C03661=1165.094,157.348,-57.134,-178.430,6.708,148.774
C03662=1165.089,157.596,-57.156,-178.428,6.710,148.774
C03663=1165.084,157.866,-57.179,-178.425,6.712,148.774
C03664=1165.079,158.135,-57.202,-178.422,6.714,148.773
C03665=1165.073,158.404,-57.226,-178.419,6.716,148.773
C03666=1165.069,158.672,-57.249,-178.416,6.718,148.772
C03667=1165.064,158.922,-57.270,-178.414,6.720,148.772
C03668=1165.059,159.170,-57.292,-178.411,6.721,148.772
C03669=1165.055,159.420,-57.314,-178.408,6.723,148.771
C03670=1165.050,159.668,-57.335,-178.405,6.725,148.771
C03671=1165.045,159.918,-57.356,-178.403,6.727,148.771
C03672=1165.040,160.167,-57.378,-178.399,6.729,148.770
C03673=1165.035,160.416,-57.400,-178.397,6.731,148.770
C03674=1165.031,160.664,-57.422,-178.395,6.733,148.770
C03675=1165.026,160.914,-57.444,-178.392,6.735,148.769
C03676=1165.021,161.163,-57.465,-178.389,6.737,148.769
C03677=1165.017,161.412,-57.487,-178.386,6.738,148.769
C03678=1165.012,161.661,-57.509,-178.384,6.740,148.768
C03679=1165.007,161.909,-57.530,-178.381,6.742,148.768
C03680=1165.003,162.159,-57.552,-178.378,6.744,148.767
C03681=1164.998,162.407,-57.574,-178.375,6.746,148.767
C03682=1164.994,162.657,-57.596,-178.372,6.748,148.767
C03683=1164.989,162.906,-57.617,-178.370,6.750,148.766
C03684=1164.984,163.155,-57.639,-178.367,6.751,148.766
C03685=1164.979,163.404,-57.661,-178.364,6.753,148.766
C03686=1164.975,163.653,-57.682,-178.362,6.755,148.765
C03687=1164.970,163.902,-57.704,-178.359,6.757,148.765
C03688=1164.965,164.151,-57.726,-178.357,6.759,148.765
C03689=1164.961,164.400,-57.748,-178.353,6.761,148.764
C03690=1164.956,164.649,-57.770,-178.351,6.763,148.764
C03691=1164.951,164.897,-57.792,-178.348,6.765,148.764
C03692=1164.947,165.147,-57.814,-178.345,6.767,148.763
C03693=1164.942,165.395,-57.835,-178.343,6.768,148.763
C03694=1164.937,165.645,-57.858,-178.340,6.770,148.762
C03695=1164.932,165.893,-57.880,-178.337,6.772,148.762
C03696=1164.928,166.143,-57.902,-178.335,6.775,148.762
C03697=1164.923,166.391,-57.923,-178.332,6.776,148.762
C03698=1164.919,166.641,-57.945,-178.329,6.778,148.761
C03699=1164.914,166.889,-57.967,-178.326,6.780,148.761
C03700=1164.910,167.139,-57.989,-178.324,6.782,148.760
C03701=1164.905,167.387,-58.012,-178.321,6.783,148.760
C03702=1164.900,167.636,-58.034,-178.318,6.786,148.760
C03703=1164.895,167.885,-58.056,-178.315,6.788,148.759
C03704=1164.891,168.134,-58.078,-178.313,6.790,148.759
C03705=1164.886,168.383,-58.100,-178.310,6.792,148.759
C03706=1164.881,168.633,-58.122,-178.308,6.793,148.758
C03707=1164.876,168.881,-58.144,-178.305,6.795,148.758
C03708=1164.872,169.130,-58.167,-178.302,6.798,148.758
C03709=1164.868,169.379,-58.188,-178.299,6.799,148.757
C03710=1164.863,169.628,-58.211,-178.296,6.801,148.757
C03711=1164.858,169.877,-58.233,-178.294,6.803,148.757
C03712=1164.853,170.126,-58.255,-178.291,6.805,148.757
C03713=1164.849,170.375,-58.277,-178.289,6.807,148.756
C03714=1164.844,170.624,-58.300,-178.285,6.809,148.756
C03715=1164.840,170.873,-58.322,-178.283,6.811,148.755
C03716=1164.835,171.122,-58.343,-178.280,6.813,148.755
C03717=1164.830,171.371,-58.367,-178.277,6.815,148.755
C03718=1164.825,171.620,-58.388,-178.275,6.817,148.755
C03719=1164.821,171.869,-58.411,-178.272,6.819,148.754
C03720=1164.816,172.118,-58.434,-178.269,6.821,148.754
C03721=1164.811,172.367,-58.456,-178.266,6.823,148.753
C03722=1164.807,172.616,-58.478,-178.264,6.825,148.753
C03723=1164.802,172.864,-58.501,-178.261,6.826,148.753
C03724=1164.797,173.114,-58.523,-178.258,6.829,148.753
C03725=1164.793,173.363,-58.545,-178.256,6.831,148.752
C03726=1164.788,173.611,-58.568,-178.253,6.833,148.752
C03727=1164.784,173.861,-58.590,-178.250,6.835,148.752
C03728=1164.780,174.109,-58.613,-178.248,6.836,148.751
C03729=1164.774,174.358,-58.635,-178.244,6.839,148.751
C03730=1164.770,174.608,-58.657,-178.242,6.841,148.751
C03731=1164.764,174.856,-58.680,-178.239,6.843,148.750
C03732=1164.760,175.105,-58.702,-178.237,6.845,148.750
C03733=1164.756,175.354,-58.725,-178.234,6.846,148.750
C03734=1164.751,175.603,-58.747,-178.231,6.849,148.749
C03735=1164.747,175.852,-58.770,-178.228,6.851,148.749
C03736=1164.742,176.101,-58.792,-178.226,6.853,148.749
C03737=1164.737,176.349,-58.815,-178.223,6.854,148.748
C03738=1164.732,176.599,-58.837,-178.220,6.857,148.748
C03739=1164.728,176.848,-58.860,-178.217,6.859,148.748
C03740=1164.723,177.098,-58.883,-178.214,6.861,148.747
C03741=1164.719,177.346,-58.905,-178.212,6.863,148.747
C03742=1164.714,177.595,-58.928,-178.210,6.864,148.747
C03743=1164.710,177.844,-58.951,-178.206,6.867,148.746
C03744=1164.704,178.092,-58.974,-178.204,6.869,148.746
C03745=1164.700,178.342,-58.996,-178.201,6.870,148.746
C03746=1164.695,178.591,-59.019,-178.199,6.873,148.746
C03747=1164.691,178.839,-59.042,-178.195,6.875,148.745
C03748=1164.686,179.088,-59.064,-178.193,6.877,148.745
C03749=1164.682,179.337,-59.087,-178.190,6.879,148.745
C03750=1164.677,179.587,-59.109,-178.188,6.881,148.744
C03751=1164.672,179.835,-59.132,-178.185,6.883,148.744
C03752=1164.668,180.084,-59.155,-178.182,6.885,148.744
C03753=1164.663,180.333,-59.179,-178.179,6.887,148.743
C03754=1164.659,180.582,-59.201,-178.177,6.889,148.743
C03755=1164.654,180.831,-59.224,-178.174,6.892,148.743
C03756=1164.649,181.079,-59.246,-178.171,6.893,148.742
C03757=1164.645,181.328,-59.270,-178.168,6.895,148.742
C03758=1164.640,181.578,-59.292,-178.166,6.897,148.742
C03759=1164.636,181.827,-59.315,-178.163,6.900,148.742
C03760=1164.630,182.075,-59.338,-178.160,6.902,148.741
C03761=1164.626,182.324,-59.361,-178.158,6.903,148.741
C03762=1164.621,182.573,-59.384,-178.154,6.906,148.741
C03763=1164.617,182.822,-59.407,-178.152,6.908,148.740
C03764=1164.613,183.071,-59.430,-178.149,6.910,148.740
C03765=1164.607,183.319,-59.453,-178.147,6.912,148.740
C03766=1164.603,183.568,-59.476,-178.144,6.914,148.739
C03767=1164.598,183.838,-59.500,-178.141,6.916,148.739
C03768=1164.593,184.108,-59.525,-178.138,6.919,148.739
C03769=1164.588,184.377,-59.551,-178.135,6.921,148.739
C03770=1164.583,184.647,-59.575,-178.132,6.923,148.738
C03771=1164.578,184.896,-59.598,-178.129,6.925,148.738
C03772=1164.574,185.145,-59.622,-178.127,6.927,148.738
C03773=1164.569,185.394,-59.645,-178.124,6.930,148.737
C03774=1164.565,185.643,-59.668,-178.121,6.931,148.737
C03775=1164.560,185.892,-59.691,-178.119,6.933,148.737
C03776=1164.555,186.141,-59.715,-178.115,6.936,148.736
C03777=1164.551,186.390,-59.738,-178.113,6.938,148.736
C03778=1164.546,186.638,-59.760,-178.110,6.940,148.736
C03779=1164.541,186.887,-59.784,-178.108,6.941,148.735
C03780=1164.537,187.136,-59.807,-178.104,6.944,148.735
C03781=1164.532,187.385,-59.830,-178.102,6.946,148.735
C03782=1164.527,187.634,-59.854,-178.100,6.948,148.735
C03783=1164.523,187.883,-59.876,-178.096,6.950,148.734
C03784=1164.519,188.132,-59.900,-178.094,6.952,148.734
C03785=1164.514,188.381,-59.923,-178.091,6.954,148.734
C03786=1164.509,188.630,-59.947,-178.088,6.957,148.734
C03787=1164.505,188.878,-59.971,-178.086,6.959,148.733
C03788=1164.500,189.126,-59.994,-178.083,6.961,148.733
C03789=1164.495,189.375,-60.017,-178.080,6.963,148.733
C03790=1164.491,189.624,-60.040,-178.077,6.965,148.732
C03791=1164.486,189.873,-60.063,-178.075,6.967,148.732
C03792=1164.482,190.122,-60.086,-178.072,6.970,148.732
C03793=1164.477,190.371,-60.110,-178.069,6.971,148.732
C03794=1164.472,190.620,-60.134,-178.067,6.974,148.731
C03795=1164.468,190.869,-60.157,-178.064,6.976,148.731
C03796=1164.463,191.118,-60.181,-178.061,6.978,148.731
C03797=1164.458,191.367,-60.204,-178.058,6.980,148.730
C03798=1164.454,191.616,-60.227,-178.056,6.983,148.730
C03799=1164.449,191.864,-60.251,-178.053,6.984,148.730
C03800=1164.445,192.113,-60.275,-178.050,6.986,148.730
C03801=1164.440,192.362,-60.298,-178.047,6.989,148.729
C03802=1164.435,192.611,-60.322,-178.045,6.991,148.729
C03803=1164.431,192.860,-60.346,-178.042,6.993,148.729
C03804=1164.426,193.109,-60.369,-178.039,6.996,148.729
C03805=1164.421,193.358,-60.392,-178.037,6.997,148.728
C03806=1164.417,193.606,-60.416,-178.034,6.999,148.728
C03807=1164.412,193.855,-60.440,-178.031,7.002,148.728
C03808=1164.408,194.104,-60.464,-178.029,7.004,148.727
C03809=1164.403,194.353,-60.487,-178.026,7.006,148.727
C03810=1164.399,194.602,-60.510,-178.023,7.008,148.727
C03811=1164.394,194.850,-60.535,-178.020,7.010,148.727
C03812=1164.389,195.099,-60.558,-178.018,7.012,148.726
C03813=1164.385,195.348,-60.581,-178.015,7.015,148.726
C03814=1164.380,195.597,-60.605,-178.012,7.017,148.726
C03815=1164.376,195.846,-60.629,-178.009,7.019,148.725
C03816=1164.371,196.094,-60.653,-178.007,7.021,148.725
C03817=1164.367,196.344,-60.677,-178.004,7.023,148.725
C03818=1164.363,196.592,-60.701,-178.001,7.026,148.725
C03819=1164.358,196.841,-60.724,-177.999,7.028,148.725
C03820=1164.353,197.090,-60.749,-177.996,7.030,148.724
C03821=1164.348,197.339,-60.772,-177.993,7.033,148.724
C03822=1164.344,197.587,-60.796,-177.991,7.034,148.724
C03823=1164.339,197.836,-60.819,-177.987,7.037,148.723
C03824=1164.335,198.085,-60.843,-177.985,7.039,148.723
C03825=1164.330,198.334,-60.867,-177.982,7.041,148.723
C03826=1164.326,198.582,-60.891,-177.979,7.043,148.723
C03827=1164.321,198.832,-60.916,-177.977,7.046,148.722
C03828=1164.316,199.081,-60.939,-177.974,7.047,148.722
C03829=1164.312,199.329,-60.963,-177.971,7.050,148.722
C03830=1164.307,199.578,-60.987,-177.969,7.052,148.722
C03831=1164.303,199.827,-61.011,-177.966,7.055,148.721
C03832=1164.299,200.075,-61.035,-177.963,7.057,148.721
C03833=1164.294,200.325,-61.059,-177.961,7.058,148.721
C03834=1164.289,200.574,-61.083,-177.958,7.061,148.721
C03835=1164.285,200.822,-61.107,-177.955,7.063,148.720
C03836=1164.280,201.071,-61.131,-177.952,7.066,148.720
C03837=1164.275,201.320,-61.155,-177.950,7.068,148.720
C03838=1164.271,201.568,-61.179,-177.947,7.070,148.720
C03839=1164.267,201.817,-61.204,-177.944,7.072,148.719
C03840=1164.262,202.066,-61.227,-177.942,7.074,148.719
C03841=1164.257,202.315,-61.252,-177.938,7.077,148.719
C03842=1164.253,202.563,-61.276,-177.936,7.079,148.719
C03843=1164.248,202.812,-61.300,-177.933,7.082,148.718
C03844=1164.243,203.062,-61.324,-177.931,7.084,148.718
C03845=1164.239,203.310,-61.348,-177.928,7.086,148.718
C03846=1164.235,203.559,-61.373,-177.925,7.088,148.718
C03847=1164.229,203.807,-61.397,-177.923,7.090,148.717
C03848=1164.226,204.056,-61.422,-177.919,7.093,148.717
C03849=1164.221,204.305,-61.446,-177.917,7.095,148.717
C03850=1164.216,204.554,-61.470,-177.914,7.097,148.717
C03851=1164.211,204.803,-61.494,-177.911,7.099,148.716
C03852=1164.208,205.052,-61.518,-177.909,7.101,148.716
C03853=1164.203,205.300,-61.543,-177.906,7.104,148.716
C03854=1164.198,205.549,-61.567,-177.904,7.106,148.716
C03855=1164.194,205.797,-61.591,-177.900,7.109,148.715
C03856=1164.189,206.047,-61.616,-177.898,7.111,148.715
C03857=1164.185,206.295,-61.640,-177.895,7.113,148.715
C03858=1164.180,206.544,-61.665,-177.893,7.116,148.715
C03859=1164.175,206.792,-61.689,-177.890,7.117,148.715
C03860=1164.171,207.042,-61.714,-177.887,7.120,148.714
C03861=1164.166,207.290,-61.738,-177.885,7.122,148.714
C03862=1164.161,207.539,-61.763,-177.881,7.125,148.714
C03863=1164.157,207.788,-61.787,-177.879,7.127,148.714
C03864=1164.153,208.036,-61.811,-177.876,7.129,148.713
C03865=1164.148,208.285,-61.836,-177.874,7.131,148.713
C03866=1164.144,208.533,-61.860,-177.870,7.134,148.713
C03867=1164.139,208.783,-61.885,-177.868,7.136,148.713
C03868=1164.135,209.031,-61.909,-177.865,7.139,148.712
C03869=1164.129,209.280,-61.934,-177.863,7.141,148.712
C03870=1164.126,209.529,-61.958,-177.860,7.143,148.712
C03871=1164.121,209.799,-61.985,-177.857,7.145,148.712
C03872=1164.116,210.070,-62.012,-177.854,7.148,148.712
C03873=1164.111,210.340,-62.039,-177.851,7.151,148.711
C03874=1164.106,210.611,-62.065,-177.848,7.153,148.711
C03875=1164.101,210.860,-62.090,-177.845,7.155,148.711
C03876=1164.096,211.109,-62.115,-177.842,7.158,148.711
C03877=1164.092,211.358,-62.140,-177.840,7.160,148.710
C03878=1164.087,211.606,-62.165,-177.837,7.162,148.710
C03879=1164.083,211.854,-62.189,-177.834,7.165,148.710
C03880=1164.078,212.104,-62.214,-177.832,7.167,148.710
C03881=1164.073,212.352,-62.239,-177.829,7.170,148.710
C03882=1164.069,212.600,-62.263,-177.826,7.171,148.709
C03883=1164.065,212.850,-62.288,-177.824,7.174,148.709
C03884=1164.060,213.098,-62.313,-177.821,7.176,148.709
C03885=1164.056,213.348,-62.338,-177.818,7.179,148.709
C03886=1164.051,213.596,-62.363,-177.815,7.181,148.708
C03887=1164.047,213.845,-62.387,-177.813,7.184,148.708
C03888=1164.042,214.093,-62.412,-177.810,7.186,148.708
C03889=1164.037,214.342,-62.437,-177.807,7.189,148.708
C03890=1164.033,214.591,-62.462,-177.805,7.190,148.707
C03891=1164.028,214.839,-62.487,-177.802,7.193,148.707
C03892=1164.024,215.088,-62.512,-177.799,7.195,148.707
C03893=1164.020,215.337,-62.536,-177.796,7.198,148.707
C03894=1164.015,215.585,-62.562,-177.794,7.200,148.707
C03895=1164.010,215.834,-62.587,-177.791,7.203,148.707
C03896=1164.006,216.084,-62.612,-177.788,7.204,148.706
C03897=1164.002,216.331,-62.637,-177.785,7.207,148.706
C03898=1163.997,216.581,-62.662,-177.783,7.209,148.706
C03899=1163.992,216.829,-62.687,-177.780,7.212,148.706
C03900=1163.988,217.078,-62.712,-177.777,7.215,148.706
C03901=1163.984,217.326,-62.737,-177.775,7.217,148.705
C03902=1163.979,217.576,-62.762,-177.772,7.220,148.705
C03903=1163.974,217.824,-62.787,-177.769,7.222,148.705
C03904=1163.970,218.073,-62.812,-177.766,7.224,148.705
C03905=1163.965,218.321,-62.838,-177.764,7.226,148.704
C03906=1163.961,218.570,-62.862,-177.761,7.229,148.704
C03907=1163.956,218.818,-62.888,-177.758,7.231,148.704
C03908=1163.952,219.067,-62.913,-177.756,7.234,148.704
C03909=1163.947,219.316,-62.938,-177.753,7.236,148.704
C03910=1163.943,219.565,-62.964,-177.750,7.239,148.703
C03911=1163.938,219.814,-62.989,-177.748,7.241,148.703
C03912=1163.934,220.062,-63.014,-177.745,7.243,148.703
C03913=1163.930,220.311,-63.039,-177.742,7.246,148.703
C03914=1163.925,220.559,-63.064,-177.739,7.248,148.703
C03915=1163.921,220.808,-63.090,-177.736,7.251,148.703
C03916=1163.916,221.056,-63.115,-177.734,7.253,148.702
C03917=1163.911,221.306,-63.140,-177.731,7.256,148.702
C03918=1163.907,221.555,-63.166,-177.728,7.258,148.702
C03919=1163.902,221.803,-63.191,-177.726,7.260,148.702
C03920=1163.898,222.052,-63.217,-177.723,7.263,148.702
C03921=1163.893,222.300,-63.242,-177.720,7.265,148.701
C03922=1163.889,222.549,-63.267,-177.717,7.268,148.701
C03923=1163.885,222.798,-63.293,-177.715,7.270,148.701
C03924=1163.880,223.046,-63.318,-177.712,7.273,148.701
C03925=1163.876,223.295,-63.343,-177.710,7.275,148.701
C03926=1163.872,223.544,-63.369,-177.706,7.278,148.700
C03927=1163.867,223.792,-63.394,-177.704,7.280,148.700
C03928=1163.863,224.041,-63.420,-177.701,7.282,148.700
C03929=1163.858,224.289,-63.445,-177.698,7.285,148.700
C03930=1163.853,224.538,-63.471,-177.696,7.287,148.700
C03931=1163.849,224.787,-63.496,-177.693,7.290,148.699
C03932=1163.844,225.035,-63.521,-177.691,7.292,148.699
C03933=1163.840,225.284,-63.547,-177.687,7.295,148.699
C03934=1163.836,225.533,-63.573,-177.685,7.298,148.699
C03935=1163.830,225.781,-63.599,-177.682,7.300,148.699
C03936=1163.826,226.030,-63.625,-177.679,7.302,148.698
C03937=1163.822,226.279,-63.650,-177.677,7.304,148.698
C03938=1163.817,226.527,-63.676,-177.674,7.307,148.698
C03939=1163.813,226.776,-63.702,-177.672,7.309,148.698
C03940=1163.808,227.025,-63.727,-177.669,7.312,148.698
C03941=1163.804,227.273,-63.753,-177.666,7.315,148.698
C03942=1163.799,227.521,-63.778,-177.663,7.317,148.697
C03943=1163.795,227.770,-63.804,-177.661,7.320,148.697
C03944=1163.791,228.019,-63.830,-177.657,7.322,148.697
C03945=1163.785,228.268,-63.856,-177.655,7.325,148.697
C03946=1163.781,228.516,-63.882,-177.652,7.327,148.697
C03947=1163.777,228.765,-63.907,-177.650,7.329,148.697
C03948=1163.773,229.014,-63.933,-177.647,7.332,148.696
C03949=1163.768,229.262,-63.959,-177.644,7.335,148.696
C03950=1163.764,229.511,-63.984,-177.642,7.337,148.696
C03951=1163.759,229.760,-64.010,-177.639,7.340,148.696
C03952=1163.755,230.008,-64.037,-177.636,7.342,148.696
C03953=1163.750,230.256,-64.063,-177.633,7.345,148.696
C03954=1163.746,230.505,-64.088,-177.631,7.348,148.695
C03955=1163.741,230.754,-64.114,-177.628,7.349,148.695
C03956=1163.736,231.003,-64.140,-177.625,7.352,148.695
C03957=1163.732,231.252,-64.166,-177.622,7.355,148.695
C03958=1163.728,231.499,-64.192,-177.620,7.357,148.695
C03959=1163.723,231.748,-64.218,-177.617,7.360,148.695
C03960=1163.719,231.997,-64.244,-177.614,7.363,148.695
C03961=1163.714,232.246,-64.270,-177.611,7.365,148.694
C03962=1163.710,232.494,-64.297,-177.609,7.368,148.694
C03963=1163.706,232.742,-64.322,-177.607,7.370,148.694
C03964=1163.701,232.991,-64.348,-177.603,7.372,148.694
C03965=1163.696,233.240,-64.374,-177.601,7.375,148.694
C03966=1163.692,233.488,-64.401,-177.598,7.377,148.694
C03967=1163.687,233.737,-64.427,-177.595,7.380,148.693
C03968=1163.683,233.986,-64.453,-177.592,7.383,148.693
C03969=1163.679,234.234,-64.479,-177.590,7.385,148.693
C03970=1163.674,234.483,-64.505,-177.587,7.388,148.693
C03971=1163.670,234.732,-64.531,-177.584,7.391,148.693
C03972=1163.666,234.980,-64.557,-177.582,7.393,148.693
C03973=1163.661,235.229,-64.584,-177.579,7.396,148.692
C03974=1163.657,235.477,-64.610,-177.576,7.398,148.692
C03975=1163.651,235.749,-64.639,-177.573,7.401,148.692
C03976=1163.647,236.021,-64.667,-177.570,7.404,148.692
C03977=1163.642,236.293,-64.696,-177.567,7.407,148.692
C03978=1163.637,236.564,-64.725,-177.564,7.410,148.692
C03979=1163.633,236.813,-64.751,-177.562,7.412,148.691
C03980=1163.628,237.061,-64.778,-177.559,7.415,148.691
C03981=1163.624,237.310,-64.803,-177.556,7.418,148.691
C03982=1163.619,237.558,-64.830,-177.554,7.420,148.691
C03983=1163.615,237.807,-64.856,-177.551,7.422,148.691
C03984=1163.610,238.055,-64.883,-177.548,7.425,148.691
C03985=1163.606,238.304,-64.909,-177.545,7.428,148.691
C03986=1163.602,238.552,-64.935,-177.543,7.430,148.691
C03987=1163.597,238.801,-64.962,-177.540,7.433,148.690
C03988=1163.593,239.050,-64.988,-177.537,7.436,148.690
C03989=1163.588,239.298,-65.015,-177.535,7.438,148.690
C03990=1163.583,239.547,-65.041,-177.532,7.441,148.690
C03991=1163.579,239.795,-65.068,-177.529,7.444,148.690
C03992=1163.575,240.044,-65.095,-177.527,7.446,148.690
C03993=1163.570,240.293,-65.121,-177.524,7.449,148.690
C03994=1163.566,240.541,-65.148,-177.521,7.452,148.689
C03995=1163.562,240.789,-65.174,-177.518,7.453,148.689
C03996=1163.557,241.039,-65.201,-177.516,7.456,148.689
C03997=1163.553,241.287,-65.227,-177.513,7.459,148.689
C03998=1163.548,241.535,-65.254,-177.510,7.462,148.689
C03999=1163.544,241.784,-65.281,-177.508,7.464,148.689
C04000=1163.539,242.033,-65.307,-177.505,7.467,148.689
C04001=1163.535,242.281,-65.334,-177.502,7.470,148.688
C04002=1163.531,242.529,-65.360,-177.500,7.472,148.688
C04003=1163.526,242.778,-65.387,-177.497,7.475,148.688
C04004=1163.521,243.027,-65.414,-177.494,7.478,148.688
C04005=1163.517,243.275,-65.440,-177.491,7.480,148.688
C04006=1163.513,243.524,-65.467,-177.489,7.483,148.688
C04007=1163.508,243.772,-65.494,-177.486,7.486,148.688
C04008=1163.504,244.020,-65.521,-177.483,7.489,148.688
C04009=1163.499,244.269,-65.548,-177.480,7.491,148.687
C04010=1163.495,244.517,-65.575,-177.478,7.493,148.687
C04011=1163.491,244.766,-65.601,-177.475,7.496,148.687
C04012=1163.486,245.014,-65.628,-177.472,7.499,148.687
C04013=1163.482,245.264,-65.655,-177.470,7.501,148.687
C04014=1163.478,245.512,-65.682,-177.467,7.504,148.687
C04015=1163.473,245.760,-65.709,-177.464,7.507,148.687
C04016=1163.469,246.009,-65.736,-177.461,7.510,148.687
C04017=1163.464,246.257,-65.763,-177.459,7.512,148.687
C04018=1163.460,246.506,-65.789,-177.456,7.515,148.686
C04019=1163.455,246.754,-65.816,-177.454,7.518,148.686
C04020=1163.451,247.003,-65.843,-177.450,7.520,148.686
C04021=1163.446,247.251,-65.871,-177.448,7.523,148.686
C04022=1163.443,247.500,-65.897,-177.446,7.526,148.686
C04023=1163.438,247.748,-65.924,-177.443,7.528,148.686
C04024=1163.433,247.997,-65.951,-177.440,7.531,148.686
C04025=1163.429,248.245,-65.979,-177.438,7.534,148.686
C04026=1163.424,248.494,-66.006,-177.435,7.536,148.685
C04027=1163.420,248.742,-66.032,-177.432,7.539,148.685
C04028=1163.416,248.990,-66.060,-177.429,7.542,148.685
C04029=1163.412,249.239,-66.087,-177.427,7.544,148.685
C04030=1163.407,249.488,-66.114,-177.424,7.547,148.685
C04031=1163.402,249.736,-66.141,-177.421,7.550,148.685
C04032=1163.398,249.985,-66.168,-177.419,7.553,148.685
C04033=1163.393,250.233,-66.196,-177.415,7.556,148.685
C04034=1163.389,250.482,-66.223,-177.413,7.558,148.685
C04035=1163.385,250.730,-66.250,-177.410,7.561,148.685
C04036=1163.381,250.978,-66.277,-177.408,7.564,148.684
C04037=1163.376,251.227,-66.304,-177.405,7.567,148.684
C04038=1163.372,251.475,-66.331,-177.403,7.569,148.684
C04039=1163.368,251.724,-66.359,-177.400,7.572,148.684
C04040=1163.363,251.972,-66.387,-177.397,7.575,148.684
C04041=1163.358,252.221,-66.414,-177.394,7.577,148.684
C04042=1163.354,252.469,-66.441,-177.391,7.580,148.684
C04043=1163.349,252.717,-66.468,-177.389,7.582,148.684
C04044=1163.345,252.967,-66.496,-177.386,7.585,148.684
C04045=1163.341,253.215,-66.523,-177.383,7.588,148.684
C04046=1163.336,253.463,-66.551,-177.381,7.591,148.684
C04047=1163.332,253.711,-66.578,-177.378,7.594,148.683
C04048=1163.328,253.961,-66.605,-177.376,7.596,148.683
C04049=1163.323,254.208,-66.633,-177.373,7.599,148.683
C04050=1163.319,254.457,-66.660,-177.370,7.602,148.683
C04051=1163.315,254.706,-66.688,-177.367,7.605,148.683
C04052=1163.310,254.954,-66.715,-177.364,7.608,148.683
C04053=1163.306,255.203,-66.742,-177.362,7.610,148.683
C04054=1163.301,255.450,-66.770,-177.359,7.613,148.683
C04055=1163.297,255.700,-66.797,-177.357,7.616,148.683
C04056=1163.293,255.947,-66.825,-177.354,7.619,148.683
C04057=1163.288,256.196,-66.852,-177.351,7.622,148.683
C04058=1163.284,256.445,-66.880,-177.349,7.624,148.682
C04059=1163.280,256.693,-66.908,-177.346,7.627,148.682
C04060=1163.275,256.941,-66.936,-177.343,7.630,148.682
C04061=1163.271,257.190,-66.963,-177.341,7.633,148.682
C04062=1163.266,257.438,-66.991,-177.338,7.636,148.682
C04063=1163.262,257.686,-67.019,-177.336,7.638,148.682
C04064=1163.258,257.935,-67.046,-177.333,7.641,148.682
C04065=1163.254,258.183,-67.074,-177.330,7.644,148.682
C04066=1163.249,258.432,-67.101,-177.327,7.647,148.682
C04067=1163.245,258.680,-67.129,-177.325,7.650,148.682
C04068=1163.240,258.928,-67.158,-177.322,7.653,148.682
C04069=1163.235,259.177,-67.185,-177.319,7.654,148.682
C04070=1163.232,259.426,-67.213,-177.316,7.657,148.681
C04071=1163.227,259.673,-67.241,-177.314,7.660,148.681
C04072=1163.223,259.923,-67.268,-177.311,7.663,148.681
C04073=1163.218,260.171,-67.296,-177.308,7.666,148.681
C04074=1163.214,260.419,-67.324,-177.305,7.669,148.681
C04075=1163.210,260.668,-67.352,-177.303,7.671,148.681
C04076=1163.205,260.916,-67.379,-177.300,7.674,148.681
C04077=1163.201,261.165,-67.408,-177.298,7.677,148.681
C04078=1163.197,261.413,-67.436,-177.295,7.680,148.681
C04079=1163.192,261.686,-67.467,-177.292,7.683,148.681
C04080=1163.187,261.959,-67.497,-177.289,7.686,148.681
C04081=1163.183,262.233,-67.528,-177.286,7.690,148.681
C04082=1163.178,262.506,-67.559,-177.283,7.693,148.681
C04083=1163.173,262.754,-67.587,-177.280,7.696,148.681
C04084=1163.168,263.002,-67.615,-177.278,7.699,148.681
C04085=1163.165,263.250,-67.643,-177.276,7.701,148.681
C04086=1163.160,263.499,-67.670,-177.273,7.704,148.681
C04087=1163.156,263.748,-67.699,-177.270,7.707,148.680
C04088=1163.151,263.996,-67.727,-177.267,7.710,148.680
C04089=1163.147,264.245,-67.755,-177.264,7.713,148.680
C04090=1163.142,264.493,-67.783,-177.262,7.716,148.680
C04091=1163.139,264.741,-67.811,-177.259,7.719,148.680
C04092=1163.134,264.989,-67.840,-177.257,7.721,148.680
C04093=1163.130,265.238,-67.868,-177.254,7.724,148.680
C04094=1163.125,265.486,-67.896,-177.251,7.727,148.680
C04095=1163.121,265.735,-67.924,-177.249,7.730,148.680
C04096=1163.117,265.982,-67.952,-177.246,7.733,148.680
C04097=1163.112,266.231,-67.981,-177.243,7.735,148.680
C04098=1163.108,266.479,-68.008,-177.240,7.738,148.680
C04099=1163.103,266.728,-68.037,-177.237,7.741,148.680
C04100=1163.099,266.976,-68.065,-177.235,7.744,148.680
C04101=1163.094,267.225,-68.094,-177.233,7.747,148.680
C04102=1163.090,267.473,-68.122,-177.230,7.750,148.680
C04103=1163.086,267.722,-68.150,-177.227,7.753,148.680
C04104=1163.082,267.970,-68.178,-177.225,7.756,148.680
C04105=1163.077,268.218,-68.207,-177.222,7.759,148.680
C04106=1163.073,268.466,-68.236,-177.219,7.762,148.680
C04107=1163.068,268.715,-68.264,-177.216,7.765,148.680
C04108=1163.064,268.963,-68.292,-177.214,7.767,148.679
C04109=1163.059,269.211,-68.321,-177.212,7.770,148.679
C04110=1163.056,269.460,-68.349,-177.209,7.773,148.679
C04111=1163.051,269.709,-68.377,-177.206,7.776,148.679
C04112=1163.047,269.956,-68.406,-177.203,7.779,148.679
C04113=1163.043,270.205,-68.435,-177.200,7.781,148.679
C04114=1163.038,270.453,-68.462,-177.198,7.784,148.679
C04115=1163.034,270.702,-68.491,-177.195,7.788,148.679
C04116=1163.030,270.950,-68.521,-177.193,7.791,148.679
C04117=1163.025,271.198,-68.548,-177.190,7.794,148.679
C04118=1163.021,271.447,-68.577,-177.188,7.796,148.679
C04119=1163.016,271.695,-68.605,-177.185,7.799,148.679
C04120=1163.012,271.943,-68.634,-177.182,7.802,148.679
C04121=1163.008,272.192,-68.663,-177.179,7.805,148.679
C04122=1163.003,272.440,-68.691,-177.177,7.808,148.679
C04123=1162.999,272.688,-68.720,-177.174,7.811,148.679
C04124=1162.995,272.937,-68.749,-177.172,7.814,148.679
C04125=1162.991,273.184,-68.778,-177.169,7.817,148.679
C04126=1162.986,273.433,-68.806,-177.166,7.820,148.679
C04127=1162.982,273.682,-68.835,-177.163,7.823,148.679
C04128=1162.978,273.929,-68.864,-177.161,7.826,148.679
C04129=1162.973,274.178,-68.892,-177.158,7.829,148.679
C04130=1162.969,274.426,-68.922,-177.156,7.831,148.679
C04131=1162.965,274.675,-68.950,-177.153,7.834,148.679
C04132=1162.960,274.922,-68.979,-177.151,7.837,148.679
C04133=1162.956,275.171,-69.008,-177.148,7.840,148.679
C04134=1162.952,275.420,-69.037,-177.145,7.843,148.679
C04135=1162.947,275.667,-69.065,-177.142,7.846,148.679
C04136=1162.943,275.916,-69.094,-177.140,7.849,148.679
C04137=1162.939,276.165,-69.123,-177.137,7.852,148.679
C04138=1162.935,276.413,-69.153,-177.135,7.855,148.679
C04139=1162.930,276.661,-69.180,-177.132,7.858,148.679
C04140=1162.926,276.909,-69.210,-177.129,7.861,148.679
C04141=1162.922,277.157,-69.239,-177.126,7.864,148.679
C04142=1162.917,277.406,-69.268,-177.124,7.867,148.679
C04143=1162.913,277.654,-69.297,-177.121,7.870,148.679
C04144=1162.909,277.902,-69.326,-177.119,7.872,148.679
C04145=1162.905,278.151,-69.355,-177.116,7.875,148.679
C04146=1162.900,278.399,-69.384,-177.114,7.878,148.679
C04147=1162.896,278.647,-69.414,-177.111,7.881,148.679
C04148=1162.891,278.895,-69.442,-177.108,7.884,148.678
C04149=1162.887,279.144,-69.471,-177.105,7.887,148.678
C04150=1162.883,279.392,-69.501,-177.103,7.890,148.679
C04151=1162.879,279.640,-69.529,-177.100,7.893,148.679
C04152=1162.875,279.889,-69.558,-177.097,7.896,148.679
C04153=1162.870,280.136,-69.588,-177.095,7.899,148.678
C04154=1162.866,280.384,-69.617,-177.092,7.902,148.678
C04155=1162.861,280.633,-69.646,-177.090,7.906,148.679
C04156=1162.857,280.882,-69.675,-177.087,7.909,148.679
C04157=1162.853,281.130,-69.705,-177.084,7.911,148.679
C04158=1162.849,281.378,-69.734,-177.081,7.914,148.678
C04159=1162.844,281.626,-69.763,-177.079,7.918,148.679
C04160=1162.840,281.874,-69.793,-177.076,7.921,148.679
C04161=1162.835,282.123,-69.821,-177.074,7.924,148.679
C04162=1162.831,282.371,-69.851,-177.071,7.927,148.679
C04163=1162.827,282.619,-69.880,-177.068,7.930,148.678
C04164=1162.823,282.868,-69.910,-177.066,7.933,148.679
C04165=1162.819,283.116,-69.939,-177.063,7.936,148.679
C04166=1162.814,283.364,-69.968,-177.060,7.939,148.679
C04167=1162.810,283.612,-69.998,-177.057,7.942,148.679
C04168=1162.806,283.860,-70.027,-177.055,7.945,148.679
C04169=1162.801,284.108,-70.057,-177.052,7.948,148.679
C04170=1162.797,284.357,-70.086,-177.050,7.950,148.679
C04171=1162.793,284.605,-70.116,-177.048,7.953,148.679
C04172=1162.789,284.853,-70.145,-177.045,7.956,148.679
C04173=1162.785,285.101,-70.174,-177.042,7.959,148.679
C04174=1162.781,285.350,-70.204,-177.040,7.962,148.679
C04175=1162.776,285.598,-70.233,-177.037,7.965,148.679
C04176=1162.771,285.847,-70.263,-177.035,7.969,148.679
C04177=1162.767,286.095,-70.293,-177.032,7.971,148.679
C04178=1162.762,286.342,-70.322,-177.029,7.974,148.679
C04179=1162.758,286.591,-70.351,-177.026,7.977,148.679
C04180=1162.754,286.839,-70.381,-177.024,7.981,148.679
C04181=1162.750,287.087,-70.411,-177.021,7.984,148.679
C04182=1162.746,287.335,-70.440,-177.019,7.987,148.679
C04183=1162.741,287.610,-70.473,-177.016,7.991,148.679
C04184=1162.736,287.885,-70.506,-177.013,7.994,148.679
C04185=1162.731,288.160,-70.539,-177.010,7.997,148.679
C04186=1162.727,288.435,-70.572,-177.007,8.000,148.679
C04187=1162.723,288.683,-70.602,-177.004,8.003,148.679
C04188=1162.718,288.932,-70.631,-177.002,8.007,148.679
C04189=1162.714,289.180,-70.661,-176.999,8.010,148.679
C04190=1162.710,289.428,-70.691,-176.996,8.013,148.679
C04191=1162.706,289.676,-70.721,-176.994,8.016,148.679
C04192=1162.701,289.924,-70.750,-176.991,8.019,148.679
C04193=1162.697,290.172,-70.781,-176.989,8.022,148.679
C04194=1162.693,290.421,-70.811,-176.986,8.025,148.679
C04195=1162.688,290.669,-70.840,-176.983,8.028,148.679
C04196=1162.684,290.917,-70.870,-176.981,8.031,148.679
C04197=1162.680,291.165,-70.900,-176.978,8.034,148.679
C04198=1162.676,291.414,-70.930,-176.976,8.037,148.679
C04199=1162.672,291.662,-70.960,-176.973,8.040,148.679
C04200=1162.667,291.910,-70.990,-176.971,8.044,148.679
C04201=1162.663,292.158,-71.020,-176.968,8.046,148.679
C04202=1162.659,292.406,-71.050,-176.965,8.049,148.679
C04203=1162.654,292.655,-71.080,-176.963,8.053,148.680
C04204=1162.650,292.902,-71.110,-176.960,8.056,148.680
C04205=1162.646,293.151,-71.140,-176.957,8.059,148.679
C04206=1162.642,293.399,-71.170,-176.955,8.062,148.680
C04207=1162.637,293.647,-71.200,-176.952,8.065,148.680
C04208=1162.633,293.895,-71.230,-176.950,8.068,148.680
C04209=1162.629,294.144,-71.260,-176.947,8.072,148.680
C04210=1162.625,294.392,-71.291,-176.944,8.075,148.680
C04211=1162.621,294.640,-71.320,-176.941,8.078,148.680
C04212=1162.616,294.888,-71.351,-176.939,8.081,148.680
C04213=1162.613,295.135,-71.381,-176.936,8.084,148.680
C04214=1162.608,295.384,-71.411,-176.934,8.087,148.680
C04215=1162.604,295.632,-71.441,-176.931,8.090,148.680
C04216=1162.600,295.881,-71.472,-176.928,8.093,148.680
C04217=1162.596,296.129,-71.502,-176.926,8.097,148.680
C04218=1162.591,296.376,-71.532,-176.923,8.100,148.680
C04219=1162.587,296.625,-71.562,-176.921,8.103,148.680
C04220=1162.583,296.872,-71.592,-176.918,8.106,148.680
C04221=1162.578,297.120,-71.623,-176.915,8.109,148.680
C04222=1162.575,297.369,-71.653,-176.913,8.112,148.680
C04223=1162.570,297.617,-71.683,-176.910,8.115,148.680
C04224=1162.566,297.865,-71.714,-176.908,8.118,148.681
C04225=1162.561,298.114,-71.744,-176.905,8.121,148.681
C04226=1162.557,298.361,-71.774,-176.903,8.124,148.681
C04227=1162.553,298.610,-71.805,-176.900,8.128,148.681
C04228=1162.549,298.858,-71.836,-176.898,8.131,148.681
C04229=1162.545,299.105,-71.866,-176.895,8.134,148.681
C04230=1162.540,299.354,-71.896,-176.892,8.138,148.681
C04231=1162.536,299.602,-71.926,-176.889,8.141,148.681
C04232=1162.532,299.850,-71.957,-176.887,8.144,148.681
C04233=1162.528,300.098,-71.988,-176.884,8.147,148.681
C04234=1162.524,300.346,-72.018,-176.882,8.150,148.681
C04235=1162.519,300.594,-72.049,-176.879,8.153,148.681
C04236=1162.515,300.843,-72.079,-176.877,8.156,148.681
C04237=1162.511,301.091,-72.110,-176.874,8.159,148.681
C04238=1162.506,301.339,-72.140,-176.871,8.162,148.681
C04239=1162.502,301.586,-72.170,-176.869,8.166,148.681
C04240=1162.498,301.835,-72.202,-176.866,8.169,148.681
C04241=1162.494,302.083,-72.232,-176.864,8.172,148.682
C04242=1162.490,302.331,-72.262,-176.861,8.175,148.682
C04243=1162.486,302.579,-72.294,-176.858,8.179,148.682
C04244=1162.481,302.827,-72.324,-176.856,8.182,148.682
C04245=1162.477,303.075,-72.355,-176.853,8.185,148.682
C04246=1162.473,303.323,-72.385,-176.850,8.188,148.682
C04247=1162.469,303.572,-72.416,-176.848,8.191,148.682
C04248=1162.464,303.820,-72.447,-176.845,8.194,148.682
C04249=1162.460,304.067,-72.478,-176.843,8.198,148.682
C04250=1162.456,304.316,-72.509,-176.840,8.201,148.682
C04251=1162.452,304.564,-72.539,-176.838,8.204,148.682
C04252=1162.447,304.812,-72.570,-176.835,8.207,148.682
C04253=1162.443,305.060,-72.602,-176.833,8.210,148.682
C04254=1162.439,305.307,-72.632,-176.830,8.213,148.683
C04255=1162.435,305.555,-72.663,-176.827,8.217,148.683
C04256=1162.431,305.804,-72.694,-176.825,8.220,148.683
C04257=1162.426,306.052,-72.725,-176.822,8.223,148.683
C04258=1162.422,306.300,-72.755,-176.820,8.226,148.683
C04259=1162.418,306.548,-72.787,-176.817,8.229,148.683
C04260=1162.414,306.796,-72.817,-176.815,8.233,148.683
C04261=1162.410,307.044,-72.849,-176.812,8.236,148.683
C04262=1162.405,307.292,-72.879,-176.810,8.239,148.683
C04263=1162.401,307.540,-72.910,-176.807,8.242,148.683
C04264=1162.397,307.788,-72.942,-176.804,8.246,148.683
C04265=1162.392,308.036,-72.973,-176.802,8.249,148.684
C04266=1162.388,308.285,-73.004,-176.799,8.252,148.684
C04267=1162.384,308.532,-73.035,-176.797,8.256,148.684
C04268=1162.380,308.780,-73.066,-176.794,8.259,148.684
C04269=1162.376,309.029,-73.097,-176.792,8.262,148.684
C04270=1162.372,309.276,-73.128,-176.789,8.265,148.684
C04271=1162.368,309.525,-73.159,-176.786,8.268,148.684
C04272=1162.363,309.772,-73.190,-176.784,8.271,148.684
C04273=1162.360,310.021,-73.222,-176.781,8.275,148.684
C04274=1162.355,310.268,-73.253,-176.778,8.278,148.684
C04275=1162.351,310.516,-73.284,-176.776,8.281,148.685
C04276=1162.347,310.764,-73.315,-176.774,8.285,148.685
C04277=1162.342,311.012,-73.346,-176.771,8.288,148.685
C04278=1162.338,311.260,-73.378,-176.768,8.291,148.685
C04279=1162.334,311.508,-73.409,-176.766,8.294,148.685
C04280=1162.330,311.756,-73.440,-176.763,8.297,148.685
C04281=1162.325,312.004,-73.471,-176.760,8.301,148.685
C04282=1162.322,312.252,-73.503,-176.758,8.304,148.685
C04283=1162.317,312.500,-73.534,-176.755,8.308,148.685
C04284=1162.313,312.748,-73.566,-176.753,8.311,148.685
C04285=1162.309,312.996,-73.596,-176.750,8.314,148.686
C04286=1162.305,313.244,-73.628,-176.748,8.317,148.686
C04287=1162.300,313.521,-73.664,-176.745,8.321,148.686
C04288=1162.296,313.799,-73.699,-176.742,8.325,148.686
C04289=1162.291,314.076,-73.734,-176.739,8.328,148.686
C04290=1162.286,314.353,-73.769,-176.736,8.332,148.686
C04291=1162.282,314.601,-73.801,-176.734,8.335,148.686
C04292=1162.277,314.849,-73.832,-176.731,8.338,148.686
C04293=1162.274,315.097,-73.863,-176.729,8.341,148.686
C04294=1162.270,315.345,-73.895,-176.726,8.345,148.687
C04295=1162.266,315.592,-73.927,-176.723,8.349,148.687
C04296=1162.261,315.841,-73.958,-176.721,8.352,148.687
C04297=1162.257,316.089,-73.990,-176.718,8.355,148.687
C04298=1162.253,316.337,-74.022,-176.716,8.358,148.687
C04299=1162.249,316.585,-74.053,-176.713,8.361,148.687
C04300=1162.245,316.833,-74.084,-176.711,8.365,148.687
C04301=1162.241,317.081,-74.116,-176.708,8.368,148.687
C04302=1162.236,317.328,-74.148,-176.705,8.372,148.688
C04303=1162.232,317.577,-74.180,-176.703,8.375,148.688
C04304=1162.228,317.825,-74.211,-176.700,8.378,148.688
C04305=1162.224,318.073,-74.243,-176.698,8.381,148.688
C04306=1162.220,318.321,-74.275,-176.696,8.384,148.688
C04307=1162.215,318.568,-74.307,-176.692,8.388,148.688
C04308=1162.211,318.816,-74.338,-176.690,8.392,148.688
C04309=1162.208,319.064,-74.370,-176.688,8.395,148.689
C04310=1162.203,319.312,-74.402,-176.685,8.398,148.689
C04311=1162.199,319.560,-74.434,-176.683,8.401,148.689
C04312=1162.195,319.808,-74.466,-176.680,8.404,148.689
C04313=1162.191,320.055,-74.498,-176.677,8.408,148.689
C04314=1162.186,320.304,-74.529,-176.675,8.411,148.689
C04315=1162.182,320.552,-74.561,-176.673,8.415,148.689
C04316=1162.178,320.800,-74.593,-176.670,8.418,148.689
C04317=1162.174,321.048,-74.625,-176.667,8.421,148.690
C04318=1162.170,321.296,-74.657,-176.665,8.424,148.690
C04319=1162.166,321.544,-74.689,-176.662,8.428,148.690
C04320=1162.162,321.791,-74.722,-176.660,8.431,148.690
C04321=1162.158,322.039,-74.753,-176.657,8.435,148.690
C04322=1162.154,322.287,-74.785,-176.655,8.438,148.690
C04323=1162.149,322.535,-74.817,-176.652,8.441,148.690
C04324=1162.145,322.783,-74.849,-176.649,8.445,148.691
C04325=1162.142,323.031,-74.881,-176.647,8.448,148.691
C04326=1162.137,323.279,-74.913,-176.644,8.451,148.691
C04327=1162.133,323.527,-74.945,-176.642,8.455,148.691
C04328=1162.128,323.775,-74.977,-176.640,8.458,148.691
C04329=1162.125,324.022,-75.010,-176.636,8.462,148.691
C04330=1162.121,324.271,-75.042,-176.634,8.465,148.691
C04331=1162.116,324.518,-75.074,-176.632,8.468,148.692
C04332=1162.113,324.766,-75.106,-176.629,8.472,148.692
C04333=1162.108,325.014,-75.138,-176.627,8.474,148.692
C04334=1162.105,325.262,-75.171,-176.624,8.479,148.692
C04335=1162.100,325.510,-75.203,-176.622,8.482,148.692
C04336=1162.096,325.758,-75.235,-176.619,8.485,148.692
C04337=1162.092,326.006,-75.267,-176.617,8.488,148.692
C04338=1162.088,326.253,-75.300,-176.614,8.492,148.693
C04339=1162.084,326.502,-75.332,-176.611,8.496,148.693
C04340=1162.079,326.749,-75.364,-176.609,8.499,148.693
C04341=1162.075,326.997,-75.397,-176.606,8.502,148.693
C04342=1162.071,327.245,-75.429,-176.604,8.505,148.693
C04343=1162.067,327.493,-75.461,-176.601,8.509,148.694
C04344=1162.063,327.741,-75.494,-176.599,8.512,148.694
C04345=1162.059,327.989,-75.526,-176.597,8.516,148.694
C04346=1162.055,328.236,-75.559,-176.594,8.519,148.694
C04347=1162.051,328.484,-75.591,-176.591,8.523,148.694
C04348=1162.046,328.732,-75.623,-176.589,8.526,148.694
C04349=1162.042,328.980,-75.656,-176.586,8.529,148.695
C04350=1162.039,329.228,-75.688,-176.584,8.533,148.695
C04351=1162.034,329.476,-75.721,-176.581,8.536,148.695
C04352=1162.030,329.724,-75.754,-176.578,8.540,148.695
C04353=1162.026,329.971,-75.786,-176.576,8.543,148.695
C04354=1162.022,330.219,-75.818,-176.574,8.546,148.695
C04355=1162.017,330.467,-75.851,-176.572,8.550,148.696
C04356=1162.014,330.715,-75.883,-176.568,8.553,148.696
C04357=1162.010,330.963,-75.916,-176.566,8.557,148.696
C04358=1162.005,331.210,-75.950,-176.564,8.560,148.696
C04359=1162.002,331.459,-75.981,-176.561,8.563,148.696
C04360=1161.998,331.706,-76.015,-176.558,8.567,148.696
C04361=1161.993,331.955,-76.047,-176.556,8.571,148.697
C04362=1161.989,332.202,-76.080,-176.553,8.574,148.697
C04363=1161.985,332.449,-76.112,-176.551,8.577,148.697
C04364=1161.981,332.697,-76.145,-176.548,8.581,148.697
C04365=1161.976,332.945,-76.178,-176.546,8.584,148.697
C04366=1161.972,333.193,-76.211,-176.544,8.588,148.698
C04367=1161.969,333.441,-76.243,-176.541,8.591,148.698
C04368=1161.964,333.689,-76.276,-176.538,8.595,148.698
C04369=1161.960,333.936,-76.309,-176.536,8.598,148.698
C04370=1161.956,334.184,-76.342,-176.533,8.601,148.698
C04371=1161.952,334.432,-76.374,-176.530,8.605,148.698
C04372=1161.948,334.680,-76.407,-176.528,8.609,148.699
C04373=1161.944,334.928,-76.441,-176.526,8.612,148.699
C04374=1161.940,335.175,-76.474,-176.524,8.615,148.699
C04375=1161.936,335.424,-76.506,-176.521,8.619,148.699
C04376=1161.931,335.671,-76.539,-176.518,8.623,148.700
C04377=1161.928,335.919,-76.572,-176.516,8.626,148.700
C04378=1161.924,336.167,-76.605,-176.514,8.629,148.700
C04379=1161.920,336.414,-76.638,-176.511,8.633,148.700
C04380=1161.916,336.662,-76.671,-176.508,8.636,148.700
C04381=1161.911,336.910,-76.705,-176.506,8.640,148.700
C04382=1161.907,337.157,-76.738,-176.503,8.644,148.701
C04383=1161.903,337.406,-76.770,-176.501,8.647,148.701
C04384=1161.899,337.654,-76.803,-176.498,8.650,148.701
C04385=1161.895,337.901,-76.836,-176.496,8.654,148.701
C04386=1161.890,338.149,-76.870,-176.493,8.658,148.701
C04387=1161.887,338.396,-76.902,-176.491,8.661,148.702
C04388=1161.883,338.644,-76.935,-176.489,8.664,148.702
C04389=1161.879,338.892,-76.968,-176.486,8.668,148.702
C04390=1161.875,339.140,-77.002,-176.483,8.672,148.702
C04391=1161.871,339.420,-77.040,-176.481,8.676,148.703
C04392=1161.866,339.699,-77.077,-176.478,8.680,148.703
C04393=1161.861,339.979,-77.115,-176.475,8.684,148.703
C04394=1161.857,340.259,-77.152,-176.473,8.687,148.703
C04395=1161.852,340.507,-77.186,-176.470,8.691,148.704
C04396=1161.848,340.754,-77.219,-176.467,8.695,148.704
C04397=1161.844,341.002,-77.252,-176.465,8.698,148.704
C04398=1161.840,341.250,-77.285,-176.462,8.702,148.704
C04399=1161.836,341.497,-77.319,-176.459,8.705,148.704
C04400=1161.832,341.745,-77.352,-176.457,8.708,148.704
C04401=1161.828,341.993,-77.386,-176.454,8.712,148.705
C04402=1161.824,342.241,-77.419,-176.452,8.716,148.705
C04403=1161.820,342.489,-77.452,-176.450,8.719,148.705
C04404=1161.816,342.736,-77.486,-176.447,8.723,148.706
C04405=1161.812,342.983,-77.519,-176.445,8.727,148.706
C04406=1161.808,343.231,-77.552,-176.443,8.730,148.706
C04407=1161.803,343.479,-77.586,-176.440,8.734,148.706
C04408=1161.800,343.727,-77.620,-176.437,8.737,148.706
C04409=1161.795,343.975,-77.654,-176.435,8.741,148.707
C04410=1161.791,344.222,-77.687,-176.432,8.745,148.707
C04411=1161.787,344.470,-77.720,-176.430,8.748,148.707
C04412=1161.783,344.717,-77.754,-176.428,8.751,148.707
C04413=1161.778,344.965,-77.787,-176.425,8.755,148.708
C04414=1161.775,345.214,-77.821,-176.422,8.759,148.708
C04415=1161.771,345.461,-77.855,-176.420,8.762,148.708
C04416=1161.767,345.709,-77.888,-176.417,8.766,148.708
C04417=1161.763,345.956,-77.922,-176.415,8.769,148.708
C04418=1161.758,346.204,-77.956,-176.413,8.773,148.709
C04419=1161.755,346.452,-77.990,-176.410,8.777,148.709
C04420=1161.751,346.699,-78.023,-176.408,8.780,148.709
C04421=1161.747,346.947,-78.056,-176.405,8.783,148.709
C04422=1161.742,347.194,-78.091,-176.403,8.788,148.710
C04423=1161.739,347.443,-78.124,-176.400,8.791,148.710
C04424=1161.735,347.690,-78.158,-176.398,8.794,148.710
C04425=1161.730,347.938,-78.192,-176.395,8.799,148.711
C04426=1161.726,348.185,-78.226,-176.393,8.802,148.711
C04427=1161.723,348.433,-78.260,-176.390,8.806,148.711
C04428=1161.718,348.681,-78.294,-176.388,8.809,148.711
C04429=1161.714,348.928,-78.328,-176.386,8.813,148.711
C04430=1161.710,349.176,-78.361,-176.383,8.817,148.712
C04431=1161.706,349.424,-78.396,-176.381,8.820,148.712
C04432=1161.702,349.672,-78.429,-176.378,8.824,148.712
C04433=1161.698,349.919,-78.463,-176.376,8.828,148.713
C04434=1161.694,350.167,-78.497,-176.373,8.831,148.713
C04435=1161.690,350.415,-78.531,-176.370,8.835,148.713
C04436=1161.686,350.662,-78.564,-176.368,8.838,148.713
C04437=1161.682,350.910,-78.599,-176.366,8.842,148.714
C04438=1161.678,351.158,-78.632,-176.363,8.846,148.714
C04439=1161.673,351.405,-78.667,-176.361,8.849,148.714
C04440=1161.670,351.653,-78.701,-176.358,8.853,148.714
C04441=1161.666,351.900,-78.735,-176.356,8.857,148.715
C04442=1161.662,352.148,-78.769,-176.354,8.860,148.715
C04443=1161.658,352.396,-78.803,-176.351,8.864,148.715
C04444=1161.654,352.643,-78.837,-176.349,8.868,148.716
C04445=1161.650,352.890,-78.871,-176.346,8.872,148.716
C04446=1161.646,353.138,-78.906,-176.344,8.875,148.716
C04447=1161.642,353.386,-78.939,-176.341,8.878,148.716
C04448=1161.637,353.634,-78.974,-176.339,8.883,148.717
C04449=1161.634,353.881,-79.008,-176.337,8.886,148.717
C04450=1161.629,354.129,-79.042,-176.334,8.890,148.717
C04451=1161.626,354.377,-79.077,-176.331,8.893,148.717
C04452=1161.622,354.624,-79.111,-176.330,8.897,148.718
C04453=1161.618,354.871,-79.145,-176.327,8.901,148.718
C04454=1161.614,355.119,-79.180,-176.324,8.904,148.718
C04455=1161.610,355.366,-79.214,-176.322,8.909,148.719
C04456=1161.606,355.615,-79.249,-176.320,8.912,148.719
C04457=1161.602,355.862,-79.282,-176.317,8.916,148.719
C04458=1161.598,356.110,-79.317,-176.314,8.920,148.719
C04459=1161.594,356.357,-79.351,-176.312,8.923,148.720
C04460=1161.590,356.604,-79.386,-176.310,8.927,148.720
C04461=1161.586,356.852,-79.420,-176.307,8.931,148.720
C04462=1161.582,357.099,-79.454,-176.305,8.935,148.721
C04463=1161.578,357.348,-79.489,-176.303,8.938,148.721
C04464=1161.573,357.595,-79.524,-176.300,8.942,148.721
C04465=1161.570,357.843,-79.558,-176.298,8.946,148.721
C04466=1161.566,358.090,-79.592,-176.295,8.950,148.722
C04467=1161.562,358.338,-79.627,-176.293,8.953,148.722
C04468=1161.558,358.585,-79.661,-176.290,8.957,148.722
C04469=1161.554,358.834,-79.696,-176.288,8.961,148.723
C04470=1161.550,359.080,-79.730,-176.286,8.964,148.723
C04471=1161.546,359.328,-79.765,-176.283,8.968,148.723
C04472=1161.542,359.576,-79.800,-176.281,8.972,148.724
C04473=1161.539,359.823,-79.834,-176.278,8.976,148.724
C04474=1161.534,360.071,-79.868,-176.276,8.979,148.724
C04475=1161.530,360.318,-79.904,-176.273,8.984,148.725
C04476=1161.526,360.566,-79.938,-176.271,8.987,148.725
C04477=1161.523,360.814,-79.973,-176.268,8.991,148.725
C04478=1161.519,361.061,-80.008,-176.266,8.995,148.726
C04479=1161.514,361.309,-80.043,-176.263,8.999,148.726
C04480=1161.510,361.557,-80.078,-176.261,9.002,148.726
C04481=1161.507,361.804,-80.111,-176.259,9.007,148.727
C04482=1161.503,362.051,-80.147,-176.256,9.010,148.727
C04483=1161.498,362.299,-80.181,-176.254,9.014,148.727
C04484=1161.495,362.546,-80.217,-176.252,9.018,148.728
C04485=1161.491,362.794,-80.251,-176.249,9.022,148.728
C04486=1161.487,363.041,-80.286,-176.247,9.025,148.728
C04487=1161.483,363.289,-80.321,-176.244,9.030,148.729
C04488=1161.479,363.536,-80.356,-176.242,9.033,148.729
C04489=1161.475,363.784,-80.391,-176.240,9.037,148.729
C04490=1161.471,364.032,-80.426,-176.237,9.041,148.730
C04491=1161.467,364.279,-80.460,-176.235,9.045,148.730
C04492=1161.463,364.527,-80.495,-176.233,9.048,148.730
C04493=1161.459,364.774,-80.530,-176.230,9.053,148.731
C04494=1161.455,365.021,-80.566,-176.228,9.056,148.731
C04495=1161.451,365.304,-80.605,-176.225,9.061,148.731
C04496=1161.446,365.586,-80.646,-176.222,9.066,148.732
C04497=1161.442,365.869,-80.686,-176.220,9.070,148.732
C04498=1161.438,366.152,-80.726,-176.217,9.074,148.733
C04499=1161.433,366.399,-80.760,-176.215,9.078,148.733
C04500=1161.430,366.647,-80.796,-176.213,9.082,148.734
C04501=1161.426,366.895,-80.831,-176.210,9.086,148.734
C04502=1161.422,367.142,-80.866,-176.208,9.090,148.734
C04503=1161.418,367.389,-80.901,-176.206,9.094,148.735
C04504=1161.414,367.637,-80.936,-176.204,9.098,148.735
C04505=1161.410,367.884,-80.971,-176.202,9.102,148.736
C04506=1161.406,368.132,-81.007,-176.200,9.105,148.736
C04507=1161.402,368.380,-81.042,-176.197,9.109,148.736
C04508=1161.398,368.627,-81.077,-176.195,9.113,148.737
C04509=1161.394,368.874,-81.112,-176.193,9.117,148.737
C04510=1161.390,369.122,-81.148,-176.191,9.121,148.738
C04511=1161.386,369.369,-81.182,-176.189,9.125,148.738
C04512=1161.382,369.616,-81.218,-176.187,9.129,148.739
C04513=1161.379,369.864,-81.254,-176.185,9.133,148.739
C04514=1161.375,370.111,-81.289,-176.183,9.136,148.739
C04515=1161.370,370.359,-81.325,-176.180,9.141,148.740
C04516=1161.366,370.607,-81.360,-176.178,9.144,148.740
C04517=1161.362,370.854,-81.395,-176.177,9.148,148.741
C04518=1161.359,371.102,-81.431,-176.175,9.153,148.741
C04519=1161.354,371.349,-81.466,-176.173,9.156,148.742
C04520=1161.351,371.596,-81.502,-176.171,9.160,148.742
C04521=1161.347,371.844,-81.537,-176.168,9.164,148.743
C04522=1161.343,372.091,-81.573,-176.167,9.168,148.743
C04523=1161.339,372.338,-81.608,-176.165,9.172,148.744
C04524=1161.334,372.586,-81.643,-176.163,9.175,148.744
C04525=1161.331,372.834,-81.679,-176.161,9.180,148.745
C04526=1161.327,373.081,-81.714,-176.159,9.184,148.745
C04527=1161.323,373.329,-81.750,-176.157,9.187,148.746
C04528=1161.319,373.576,-81.785,-176.156,9.191,148.746
C04529=1161.315,373.823,-81.821,-176.154,9.195,148.747
C04530=1161.311,374.071,-81.857,-176.152,9.199,148.747
C04531=1161.307,374.318,-81.892,-176.150,9.203,148.748
C04532=1161.304,374.566,-81.928,-176.149,9.207,148.749
C04533=1161.300,374.813,-81.963,-176.147,9.211,148.749
C04534=1161.296,375.060,-81.999,-176.146,9.214,148.750
C04535=1161.292,375.307,-82.035,-176.144,9.218,148.750
C04536=1161.288,375.555,-82.071,-176.143,9.222,148.751
C04537=1161.284,375.802,-82.107,-176.141,9.226,148.751
C04538=1161.281,376.050,-82.142,-176.139,9.230,148.752
C04539=1161.276,376.298,-82.178,-176.138,9.234,148.752
C04540=1161.272,376.544,-82.213,-176.136,9.237,148.753
C04541=1161.268,376.792,-82.249,-176.135,9.241,148.754
C04542=1161.265,377.039,-82.285,-176.134,9.245,148.754
C04543=1161.260,377.287,-82.321,-176.132,9.249,148.755
C04544=1161.257,377.534,-82.357,-176.131,9.253,148.756
C04545=1161.253,377.782,-82.392,-176.129,9.257,148.756
C04546=1161.249,378.029,-82.429,-176.128,9.261,148.757
C04547=1161.245,378.277,-82.464,-176.126,9.265,148.757
C04548=1161.241,378.524,-82.499,-176.125,9.268,148.758
C04549=1161.237,378.771,-82.536,-176.124,9.272,148.759
C04550=1161.233,379.018,-82.572,-176.123,9.276,148.759
C04551=1161.230,379.266,-82.607,-176.122,9.280,148.760
C04552=1161.225,379.514,-82.643,-176.121,9.283,148.761
C04553=1161.222,379.761,-82.680,-176.119,9.287,148.761
C04554=1161.218,380.008,-82.715,-176.118,9.291,148.762
C04555=1161.214,380.256,-82.751,-176.117,9.294,148.763
C04556=1161.210,380.503,-82.788,-176.116,9.298,148.763
C04557=1161.206,380.751,-82.824,-176.115,9.302,148.764
C04558=1161.202,380.997,-82.859,-176.114,9.305,148.765
C04559=1161.198,381.245,-82.895,-176.113,9.310,148.766
C04560=1161.194,381.492,-82.931,-176.112,9.313,148.766
C04561=1161.190,381.740,-82.967,-176.111,9.317,148.767
C04562=1161.186,381.987,-83.004,-176.110,9.320,148.768
C04563=1161.183,382.234,-83.039,-176.109,9.324,148.768
C04564=1161.179,382.482,-83.075,-176.109,9.328,148.769
C04565=1161.175,382.729,-83.112,-176.108,9.331,148.770
C04566=1161.171,382.977,-83.147,-176.107,9.335,148.770
C04567=1161.167,383.224,-83.183,-176.106,9.338,148.771
C04568=1161.163,383.471,-83.220,-176.106,9.342,148.772
C04569=1161.159,383.719,-83.256,-176.106,9.345,148.773
C04570=1161.156,383.966,-83.292,-176.105,9.349,148.774
C04571=1161.152,384.213,-83.328,-176.104,9.352,148.774
C04572=1161.148,384.461,-83.365,-176.103,9.356,148.775
C04573=1161.144,384.708,-83.400,-176.103,9.359,148.776
C04574=1161.140,384.955,-83.437,-176.102,9.362,148.776
C04575=1161.136,385.203,-83.472,-176.102,9.366,148.777
C04576=1161.132,385.451,-83.509,-176.102,9.369,148.778
C04577=1161.129,385.697,-83.545,-176.101,9.373,148.779
C04578=1161.124,385.945,-83.581,-176.101,9.376,148.780
C04579=1161.121,386.192,-83.617,-176.101,9.380,148.781
C04580=1161.116,386.440,-83.653,-176.101,9.382,148.781
C04581=1161.113,386.687,-83.690,-176.100,9.386,148.782
C04582=1161.109,386.935,-83.726,-176.100,9.389,148.783
C04583=1161.105,387.182,-83.762,-176.099,9.392,148.784
C04584=1161.101,387.429,-83.799,-176.100,9.395,148.784
C04585=1161.098,387.676,-83.834,-176.100,9.399,148.785
C04586=1161.094,387.923,-83.871,-176.100,9.401,148.786
C04587=1161.090,388.171,-83.907,-176.100,9.405,148.787
C04588=1161.086,388.418,-83.944,-176.100,9.407,148.788
C04589=1161.082,388.666,-83.979,-176.099,9.411,148.788
C04590=1161.078,388.913,-84.016,-176.100,9.414,148.789
C04591=1161.074,389.160,-84.052,-176.099,9.417,148.790
C04592=1161.070,389.408,-84.089,-176.100,9.420,148.791
C04593=1161.067,389.654,-84.125,-176.100,9.423,148.792
C04594=1161.062,389.902,-84.161,-176.100,9.426,148.792
C04595=1161.058,390.149,-84.198,-176.100,9.429,148.793
C04596=1161.055,390.397,-84.233,-176.100,9.431,148.794
C04597=1161.051,390.644,-84.270,-176.101,9.434,148.795
C04598=1161.047,390.891,-84.306,-176.101,9.438,148.796
C04599=1161.042,391.177,-84.348,-176.101,9.441,148.797
C04600=1161.038,391.463,-84.390,-176.101,9.444,148.798
C04601=1161.034,391.748,-84.432,-176.102,9.447,148.798
C04602=1161.029,392.034,-84.474,-176.102,9.450,148.799
C04603=1161.026,392.281,-84.510,-176.102,9.453,148.800
C04604=1161.022,392.528,-84.547,-176.103,9.455,148.801
C04605=1161.017,392.776,-84.583,-176.103,9.458,148.802
C04606=1161.014,393.023,-84.620,-176.104,9.461,148.803
C04607=1161.010,393.270,-84.656,-176.104,9.463,148.803
C04608=1161.006,393.517,-84.692,-176.104,9.466,148.804
C04609=1161.002,393.765,-84.729,-176.104,9.469,148.805
C04610=1160.998,394.012,-84.764,-176.105,9.472,148.806
C04611=1160.994,394.259,-84.801,-176.105,9.474,148.807
C04612=1160.990,394.506,-84.838,-176.106,9.476,148.807
C04613=1160.986,394.754,-84.874,-176.106,9.479,148.808
C04614=1160.982,395.001,-84.910,-176.107,9.482,148.809
C04615=1160.979,395.248,-84.947,-176.107,9.484,148.810
C04616=1160.975,395.497,-84.983,-176.108,9.486,148.811
C04617=1160.971,395.744,-85.020,-176.108,9.489,148.811
C04618=1160.968,395.991,-85.056,-176.109,9.492,148.812
C04619=1160.963,396.238,-85.092,-176.110,9.494,148.813
C04620=1160.959,396.486,-85.129,-176.110,9.496,148.814
C04621=1160.956,396.732,-85.166,-176.111,9.498,148.814
C04622=1160.952,396.980,-85.202,-176.111,9.501,148.815
C04623=1160.948,397.227,-85.238,-176.111,9.504,148.816
C04624=1160.944,397.474,-85.275,-176.112,9.505,148.817
C04625=1160.940,397.722,-85.312,-176.113,9.508,148.818
C04626=1160.936,397.969,-85.347,-176.113,9.510,148.818
C04627=1160.932,398.216,-85.384,-176.114,9.513,148.819
C04628=1160.928,398.463,-85.421,-176.115,9.515,148.820
C04629=1160.924,398.711,-85.457,-176.115,9.517,148.820
C04630=1160.920,398.958,-85.493,-176.116,9.519,148.821
C04631=1160.917,399.205,-85.530,-176.117,9.521,148.822
C04632=1160.913,399.452,-85.567,-176.117,9.524,148.823
C04633=1160.909,399.701,-85.603,-176.118,9.526,148.823
C04634=1160.906,399.948,-85.639,-176.118,9.528,148.824
C04635=1160.902,400.195,-85.676,-176.119,9.530,148.825
C04636=1160.897,400.443,-85.712,-176.120,9.532,148.826
C04637=1160.894,400.689,-85.749,-176.120,9.535,148.826
C04638=1160.890,400.937,-85.785,-176.121,9.537,148.827
C04639=1160.886,401.184,-85.822,-176.122,9.538,148.828
C04640=1160.882,401.431,-85.858,-176.122,9.541,148.829
C04641=1160.878,401.679,-85.895,-176.123,9.543,148.829
C04642=1160.875,401.925,-85.931,-176.124,9.545,148.830
C04643=1160.871,402.173,-85.968,-176.124,9.547,148.831
C04644=1160.866,402.420,-86.004,-176.125,9.549,148.831
C04645=1160.863,402.667,-86.040,-176.125,9.551,148.832
C04646=1160.859,402.914,-86.077,-176.126,9.553,148.833
C04647=1160.855,403.162,-86.114,-176.127,9.555,148.834
C04648=1160.851,403.410,-86.150,-176.127,9.557,148.834
C04649=1160.847,403.657,-86.187,-176.128,9.559,148.835
C04650=1160.843,403.904,-86.224,-176.129,9.561,148.836
C04651=1160.840,404.151,-86.260,-176.129,9.564,148.836
C04652=1160.836,404.399,-86.296,-176.130,9.565,148.837
C04653=1160.832,404.646,-86.332,-176.131,9.567,148.838
C04654=1160.828,404.893,-86.369,-176.131,9.569,148.838
C04655=1160.824,405.140,-86.406,-176.132,9.571,148.839
C04656=1160.820,405.388,-86.441,-176.133,9.572,148.840
C04657=1160.816,405.635,-86.478,-176.133,9.575,148.840
C04658=1160.812,405.882,-86.515,-176.134,9.577,148.841
C04659=1160.809,406.129,-86.551,-176.134,9.578,148.842
C04660=1160.805,406.378,-86.588,-176.135,9.580,148.842
C04661=1160.801,406.625,-86.625,-176.136,9.582,148.843
C04662=1160.798,406.872,-86.661,-176.137,9.584,148.844
C04663=1160.793,407.119,-86.698,-176.137,9.587,148.845
C04664=1160.789,407.367,-86.734,-176.138,9.588,148.845
C04665=1160.786,407.613,-86.770,-176.138,9.590,148.846
C04666=1160.782,407.861,-86.807,-176.139,9.591,148.846
C04667=1160.778,408.108,-86.844,-176.139,9.593,148.847
C04668=1160.774,408.355,-86.880,-176.140,9.595,148.848
C04669=1160.770,408.603,-86.916,-176.141,9.597,148.848
C04670=1160.766,408.850,-86.953,-176.141,9.599,148.849
C04671=1160.762,409.097,-86.990,-176.141,9.601,148.850
C04672=1160.759,409.344,-87.027,-176.142,9.603,148.850
C04673=1160.754,409.592,-87.063,-176.143,9.604,148.851
C04674=1160.751,409.839,-87.099,-176.144,9.606,148.852
C04675=1160.747,410.086,-87.136,-176.144,9.608,148.852
C04676=1160.743,410.334,-87.173,-176.145,9.610,148.853
C04677=1160.740,410.580,-87.209,-176.145,9.612,148.853
C04678=1160.735,410.828,-87.245,-176.145,9.614,148.854
C04679=1160.731,411.075,-87.282,-176.146,9.615,148.855
C04680=1160.728,411.322,-87.318,-176.147,9.617,148.855
C04681=1160.724,411.569,-87.355,-176.147,9.619,148.856
C04682=1160.719,411.817,-87.391,-176.148,9.621,148.857
C04683=1160.716,412.065,-87.428,-176.148,9.622,148.857
C04684=1160.712,412.312,-87.465,-176.149,9.624,148.858
C04685=1160.708,412.559,-87.502,-176.149,9.626,148.858
C04686=1160.705,412.806,-87.538,-176.150,9.628,148.859
C04687=1160.700,413.054,-87.574,-176.150,9.630,148.859
C04688=1160.696,413.301,-87.611,-176.151,9.631,148.860
C04689=1160.692,413.548,-87.648,-176.152,9.633,148.861
C04690=1160.689,413.795,-87.684,-176.152,9.635,148.861
C04691=1160.685,414.042,-87.721,-176.153,9.636,148.862
C04692=1160.681,414.290,-87.758,-176.153,9.639,148.863
C04693=1160.678,414.538,-87.794,-176.153,9.641,148.863
C04694=1160.674,414.785,-87.831,-176.154,9.642,148.864
C04695=1160.669,415.032,-87.868,-176.154,9.644,148.864
C04696=1160.666,415.279,-87.904,-176.155,9.646,148.865
C04697=1160.663,415.527,-87.940,-176.155,9.647,148.865
C04698=1160.661,415.774,-87.976,-176.156,9.649,148.866
C04699=1160.661,416.133,-88.029,-176.157,9.652,148.867
C04700=1160.662,416.492,-88.082,-176.157,9.654,148.868
C04701=1160.665,416.851,-88.134,-176.158,9.656,148.868
C04702=1160.669,417.210,-88.185,-176.158,9.659,148.869
C04703=1160.248,417.211,-88.232,-176.161,9.670,148.873
C04704=1160.244,416.850,-88.180,-176.160,9.667,148.872
C04705=1160.241,416.487,-88.127,-176.160,9.665,148.871
C04706=1160.240,416.126,-88.075,-176.159,9.662,148.870
C04707=1160.241,415.762,-88.021,-176.158,9.660,148.870
C04708=1160.243,415.515,-87.985,-176.158,9.658,148.869
C04709=1160.245,415.267,-87.949,-176.158,9.656,148.868
C04710=1160.249,415.020,-87.912,-176.157,9.655,148.868
C04711=1160.253,414.773,-87.876,-176.157,9.653,148.867
C04712=1160.257,414.526,-87.839,-176.156,9.651,148.867
C04713=1160.260,414.279,-87.802,-176.155,9.650,148.866
C04714=1160.264,414.031,-87.765,-176.155,9.648,148.866
C04715=1160.268,413.783,-87.729,-176.155,9.646,148.865
C04716=1160.271,413.537,-87.693,-176.154,9.644,148.864
C04717=1160.276,413.289,-87.656,-176.154,9.642,148.864
C04718=1160.280,413.042,-87.619,-176.153,9.641,148.863
C04719=1160.283,412.795,-87.583,-176.153,9.639,148.863
C04720=1160.287,412.548,-87.546,-176.152,9.637,148.862
C04721=1160.292,412.300,-87.510,-176.151,9.635,148.861
C04722=1160.296,412.053,-87.473,-176.152,9.633,148.861
C04723=1160.299,411.806,-87.437,-176.151,9.631,148.860
C04724=1160.302,411.558,-87.399,-176.150,9.630,148.859
C04725=1160.307,411.311,-87.363,-176.149,9.628,148.859
C04726=1160.310,411.064,-87.327,-176.149,9.626,148.858
C04727=1160.314,410.817,-87.290,-176.148,9.624,148.858
C04728=1160.318,410.569,-87.253,-176.148,9.623,148.857
C04729=1160.322,410.322,-87.217,-176.147,9.621,148.856
C04730=1160.326,410.075,-87.180,-176.147,9.619,148.856
C04731=1160.330,409.827,-87.144,-176.146,9.617,148.855
C04732=1160.334,409.581,-87.108,-176.146,9.615,148.854
C04733=1160.338,409.333,-87.071,-176.145,9.613,148.854
C04734=1160.342,409.086,-87.034,-176.144,9.612,148.853
C04735=1160.345,408.839,-86.997,-176.144,9.610,148.852
C04736=1160.349,408.591,-86.961,-176.143,9.608,148.852
C04737=1160.353,408.344,-86.924,-176.142,9.606,148.851
C04738=1160.356,408.097,-86.888,-176.142,9.604,148.850
C04739=1160.361,407.850,-86.851,-176.141,9.602,148.850
C04740=1160.365,407.602,-86.814,-176.141,9.600,148.849
C04741=1160.368,407.355,-86.779,-176.140,9.599,148.849
C04742=1160.372,407.108,-86.742,-176.139,9.597,148.848
C04743=1160.376,406.860,-86.705,-176.139,9.595,148.847
C04744=1160.380,406.614,-86.669,-176.138,9.593,148.847
C04745=1160.384,406.366,-86.633,-176.137,9.592,148.846
C04746=1160.388,406.118,-86.596,-176.137,9.589,148.845
C04747=1160.391,405.871,-86.559,-176.136,9.587,148.845
C04748=1160.395,405.624,-86.522,-176.136,9.586,148.844
C04749=1160.400,405.376,-86.486,-176.135,9.584,148.843
C04750=1160.403,405.129,-86.450,-176.134,9.582,148.843
C04751=1160.407,404.882,-86.413,-176.134,9.580,148.842
C04752=1160.411,404.635,-86.376,-176.133,9.578,148.841
C04753=1160.414,404.388,-86.340,-176.132,9.576,148.840
C04754=1160.419,404.140,-86.304,-176.132,9.574,148.840
C04755=1160.423,403.893,-86.267,-176.131,9.572,148.839
C04756=1160.426,403.646,-86.231,-176.130,9.570,148.839
C04757=1160.430,403.399,-86.194,-176.130,9.568,148.838
C04758=1160.434,403.150,-86.157,-176.129,9.566,148.837
C04759=1160.438,402.903,-86.121,-176.128,9.564,148.836
C04760=1160.442,402.656,-86.084,-176.128,9.562,148.836
C04761=1160.446,402.409,-86.047,-176.127,9.560,148.835
C04762=1160.449,402.162,-86.012,-176.127,9.558,148.834
C04763=1160.454,401.914,-85.975,-176.126,9.556,148.833
C04764=1160.458,401.667,-85.938,-176.125,9.554,148.833
C04765=1160.461,401.420,-85.902,-176.125,9.552,148.832
C04766=1160.465,401.172,-85.866,-176.124,9.550,148.831
C04767=1160.469,400.926,-85.830,-176.123,9.548,148.831
C04768=1160.473,400.678,-85.793,-176.123,9.545,148.830
C04769=1160.477,400.431,-85.756,-176.122,9.543,148.829
C04770=1160.481,400.184,-85.720,-176.121,9.541,148.828
C04771=1160.484,399.936,-85.683,-176.121,9.539,148.828
C04772=1160.488,399.689,-85.646,-176.120,9.537,148.827
C04773=1160.492,399.441,-85.611,-176.119,9.535,148.826
C04774=1160.496,399.194,-85.574,-176.119,9.533,148.826
C04775=1160.500,398.947,-85.537,-176.118,9.530,148.825
C04776=1160.503,398.700,-85.501,-176.118,9.528,148.824
C04777=1160.508,398.452,-85.465,-176.116,9.526,148.823
C04778=1160.511,398.205,-85.428,-176.116,9.523,148.822
C04779=1160.515,397.958,-85.391,-176.115,9.521,148.822
C04780=1160.519,397.711,-85.355,-176.115,9.519,148.821
C04781=1160.523,397.463,-85.319,-176.114,9.517,148.820
C04782=1160.527,397.216,-85.282,-176.114,9.514,148.819
C04783=1160.531,396.969,-85.245,-176.113,9.512,148.819
C04784=1160.535,396.721,-85.210,-176.113,9.509,148.818
C04785=1160.539,396.474,-85.173,-176.112,9.508,148.817
C04786=1160.542,396.227,-85.136,-176.111,9.505,148.816
C04787=1160.546,395.979,-85.100,-176.111,9.503,148.816
C04788=1160.550,395.732,-85.063,-176.110,9.500,148.815
C04789=1160.554,395.485,-85.027,-176.110,9.498,148.814
C04790=1160.558,395.238,-84.990,-176.109,9.496,148.813
C04791=1160.562,394.990,-84.954,-176.109,9.493,148.812
C04792=1160.565,394.743,-84.918,-176.108,9.490,148.811
C04793=1160.569,394.496,-84.881,-176.108,9.488,148.811
C04794=1160.573,394.248,-84.845,-176.107,9.485,148.810
C04795=1160.577,394.001,-84.808,-176.107,9.483,148.809
C04796=1160.581,393.754,-84.772,-176.106,9.480,148.808
C04797=1160.585,393.506,-84.736,-176.106,9.477,148.808
C04798=1160.589,393.259,-84.699,-176.105,9.475,148.807
C04799=1160.592,393.012,-84.663,-176.105,9.472,148.806
C04800=1160.597,392.764,-84.627,-176.105,9.469,148.805
C04801=1160.601,392.517,-84.590,-176.105,9.467,148.804
C04802=1160.604,392.270,-84.554,-176.104,9.465,148.804
C04803=1160.609,392.023,-84.518,-176.103,9.462,148.803
C04804=1160.613,391.737,-84.475,-176.103,9.458,148.802
C04805=1160.618,391.451,-84.433,-176.103,9.455,148.801
C04806=1160.621,391.166,-84.391,-176.103,9.452,148.800
C04807=1160.626,390.879,-84.349,-176.102,9.449,148.799
C04808=1160.629,390.633,-84.313,-176.102,9.446,148.798
C04809=1160.634,390.385,-84.277,-176.102,9.443,148.797
C04810=1160.637,390.138,-84.240,-176.102,9.440,148.797
C04811=1160.642,389.890,-84.204,-176.102,9.437,148.796
C04812=1160.645,389.643,-84.168,-176.101,9.434,148.795
C04813=1160.649,389.396,-84.131,-176.101,9.431,148.794
C04814=1160.653,389.149,-84.095,-176.101,9.428,148.793
C04815=1160.657,388.901,-84.059,-176.101,9.425,148.793
C04816=1160.660,388.654,-84.023,-176.101,9.422,148.792
C04817=1160.665,388.407,-83.986,-176.101,9.419,148.791
C04818=1160.669,388.159,-83.949,-176.101,9.416,148.790
C04819=1160.672,387.912,-83.914,-176.101,9.413,148.789
C04820=1160.676,387.665,-83.877,-176.101,9.410,148.788
C04821=1160.680,387.417,-83.841,-176.101,9.407,148.788
C04822=1160.684,387.170,-83.805,-176.101,9.404,148.787
C04823=1160.688,386.923,-83.769,-176.102,9.400,148.786
C04824=1160.692,386.675,-83.732,-176.102,9.396,148.785
C04825=1160.696,386.428,-83.697,-176.102,9.394,148.785
C04826=1160.700,386.181,-83.660,-176.102,9.391,148.784
C04827=1160.703,385.933,-83.624,-176.102,9.387,148.783
C04828=1160.707,385.686,-83.587,-176.103,9.384,148.782
C04829=1160.711,385.438,-83.552,-176.103,9.380,148.781
C04830=1160.715,385.191,-83.515,-176.104,9.377,148.781
C04831=1160.719,384.944,-83.479,-176.104,9.374,148.780
C04832=1160.723,384.697,-83.443,-176.105,9.370,148.779
C04833=1160.727,384.449,-83.407,-176.105,9.367,148.778
C04834=1160.731,384.202,-83.370,-176.106,9.363,148.778
C04835=1160.734,383.954,-83.335,-176.106,9.360,148.777
C04836=1160.738,383.708,-83.298,-176.106,9.357,148.776
C04837=1160.742,383.460,-83.262,-176.107,9.352,148.775
C04838=1160.745,383.213,-83.226,-176.108,9.349,148.774
C04839=1160.750,382.965,-83.190,-176.109,9.346,148.774
C04840=1160.754,382.718,-83.154,-176.109,9.343,148.773
C04841=1160.758,382.470,-83.117,-176.110,9.338,148.772
C04842=1160.761,382.223,-83.082,-176.111,9.335,148.772
C04843=1160.765,381.976,-83.045,-176.112,9.331,148.771
C04844=1160.770,381.729,-83.010,-176.113,9.328,148.770
C04845=1160.773,381.481,-82.974,-176.114,9.324,148.770
C04846=1160.777,381.234,-82.937,-176.114,9.320,148.769
C04847=1160.781,380.987,-82.902,-176.115,9.316,148.768
C04848=1160.785,380.739,-82.866,-176.116,9.313,148.767
C04849=1160.789,380.492,-82.829,-176.118,9.309,148.767
C04850=1160.792,380.244,-82.794,-176.118,9.306,148.766
C04851=1160.797,379.997,-82.758,-176.120,9.302,148.765
C04852=1160.800,379.750,-82.721,-176.121,9.298,148.765
C04853=1160.804,379.502,-82.686,-176.122,9.295,148.764
C04854=1160.808,379.254,-82.650,-176.123,9.291,148.763
C04855=1160.812,379.007,-82.614,-176.124,9.287,148.763
C04856=1160.817,378.760,-82.578,-176.125,9.283,148.762
C04857=1160.820,378.513,-82.542,-176.127,9.279,148.761
C04858=1160.824,378.265,-82.507,-176.128,9.276,148.761
C04859=1160.828,378.018,-82.470,-176.129,9.272,148.760
C04860=1160.832,377.771,-82.434,-176.131,9.268,148.759
C04861=1160.835,377.523,-82.399,-176.132,9.264,148.759
C04862=1160.839,377.276,-82.363,-176.134,9.260,148.758
C04863=1160.843,377.028,-82.327,-176.135,9.256,148.758
C04864=1160.847,376.780,-82.291,-176.136,9.252,148.757
C04865=1160.851,376.534,-82.256,-176.138,9.248,148.756
C04866=1160.855,376.286,-82.219,-176.139,9.244,148.756
C04867=1160.859,376.039,-82.184,-176.141,9.241,148.755
C04868=1160.863,375.791,-82.148,-176.143,9.237,148.755
C04869=1160.866,375.544,-82.113,-176.144,9.233,148.754
C04870=1160.871,375.296,-82.077,-176.146,9.229,148.753
C04871=1160.875,375.049,-82.041,-176.147,9.226,148.753
C04872=1160.879,374.802,-82.006,-176.149,9.222,148.752
C04873=1160.882,374.554,-81.970,-176.150,9.218,148.752
C04874=1160.887,374.307,-81.934,-176.152,9.214,148.751
C04875=1160.891,374.059,-81.899,-176.154,9.209,148.751
C04876=1160.894,373.812,-81.863,-176.156,9.206,148.750
C04877=1160.898,373.565,-81.828,-176.157,9.202,148.750
C04878=1160.902,373.317,-81.792,-176.159,9.198,148.749
C04879=1160.906,373.070,-81.757,-176.161,9.194,148.749
C04880=1160.910,372.822,-81.721,-176.163,9.190,148.748
C04881=1160.914,372.574,-81.685,-176.165,9.186,148.748
C04882=1160.918,372.328,-81.650,-176.167,9.183,148.747
C04883=1160.922,372.080,-81.614,-176.168,9.179,148.747
C04884=1160.925,371.833,-81.579,-176.171,9.175,148.746
C04885=1160.929,371.585,-81.543,-176.173,9.171,148.746
C04886=1160.933,371.338,-81.508,-176.174,9.167,148.745
C04887=1160.938,371.091,-81.472,-176.177,9.163,148.745
C04888=1160.941,370.843,-81.436,-176.179,9.159,148.744
C04889=1160.945,370.595,-81.402,-176.180,9.155,148.744
C04890=1160.949,370.347,-81.366,-176.183,9.151,148.743
C04891=1160.953,370.101,-81.331,-176.185,9.147,148.743
C04892=1160.957,369.853,-81.295,-176.187,9.144,148.742
C04893=1160.961,369.606,-81.260,-176.189,9.139,148.742
C04894=1160.965,369.357,-81.225,-176.191,9.136,148.742
C04895=1160.969,369.111,-81.190,-176.193,9.131,148.741
C04896=1160.973,368.863,-81.154,-176.195,9.128,148.741
C04897=1160.976,368.616,-81.119,-176.197,9.124,148.740
C04898=1160.981,368.368,-81.084,-176.200,9.120,148.740
C04899=1160.984,368.121,-81.049,-176.201,9.116,148.739
C04900=1160.988,367.873,-81.013,-176.204,9.112,148.739
C04901=1160.992,367.626,-80.978,-176.206,9.109,148.739
C04902=1160.996,367.378,-80.943,-176.209,9.104,148.738
C04903=1161.000,367.131,-80.908,-176.211,9.100,148.738
C04904=1161.004,366.883,-80.872,-176.212,9.097,148.737
C04905=1161.008,366.636,-80.837,-176.215,9.092,148.737
C04906=1161.012,366.388,-80.802,-176.217,9.089,148.737
C04907=1161.016,366.140,-80.767,-176.220,9.085,148.736
C04908=1161.021,365.858,-80.727,-176.222,9.080,148.736
C04909=1161.025,365.575,-80.687,-176.225,9.076,148.735
C04910=1161.029,365.293,-80.647,-176.227,9.072,148.735
C04911=1161.034,365.010,-80.607,-176.230,9.067,148.734
C04912=1161.037,364.763,-80.572,-176.233,9.063,148.734
C04913=1161.042,364.516,-80.537,-176.235,9.060,148.734
C04914=1161.046,364.268,-80.502,-176.237,9.055,148.733
C04915=1161.050,364.020,-80.467,-176.239,9.052,148.733
C04916=1161.054,363.773,-80.432,-176.242,9.048,148.733
C04917=1161.058,363.525,-80.397,-176.244,9.044,148.732
C04918=1161.062,363.278,-80.362,-176.247,9.040,148.732
C04919=1161.065,363.031,-80.327,-176.249,9.037,148.732
C04920=1161.069,362.782,-80.293,-176.251,9.032,148.731
C04921=1161.074,362.536,-80.257,-176.254,9.029,148.731
C04922=1161.077,362.287,-80.223,-176.256,9.025,148.731
C04923=1161.082,362.040,-80.188,-176.258,9.021,148.730
C04924=1161.085,361.793,-80.153,-176.261,9.017,148.730
C04925=1161.089,361.545,-80.118,-176.264,9.013,148.730
C04926=1161.094,361.297,-80.084,-176.266,9.009,148.729
C04927=1161.097,361.050,-80.048,-176.269,9.005,148.729
C04928=1161.101,360.803,-80.014,-176.271,9.002,148.729
C04929=1161.105,360.555,-79.980,-176.274,8.998,148.728
C04930=1161.109,360.308,-79.944,-176.275,8.994,148.728
C04931=1161.113,360.060,-79.910,-176.278,8.990,148.728
C04932=1161.117,359.813,-79.876,-176.281,8.987,148.727
C04933=1161.121,359.564,-79.841,-176.283,8.982,148.727
C04934=1161.125,359.318,-79.806,-176.285,8.979,148.727
C04935=1161.129,359.070,-79.771,-176.288,8.975,148.726
C04936=1161.133,358.822,-79.737,-176.290,8.971,148.726
C04937=1161.137,358.574,-79.702,-176.293,8.967,148.726
C04938=1161.141,358.327,-79.668,-176.295,8.964,148.726
C04939=1161.145,358.079,-79.633,-176.297,8.960,148.725
C04940=1161.149,357.832,-79.599,-176.300,8.956,148.725
C04941=1161.152,357.584,-79.564,-176.302,8.953,148.725
C04942=1161.157,357.337,-79.530,-176.305,8.949,148.724
C04943=1161.161,357.089,-79.495,-176.307,8.945,148.724
C04944=1161.165,356.842,-79.461,-176.310,8.941,148.724
C04945=1161.169,356.594,-79.426,-176.312,8.938,148.724
C04946=1161.173,356.347,-79.392,-176.315,8.933,148.723
C04947=1161.176,356.098,-79.357,-176.317,8.930,148.723
C04948=1161.181,355.851,-79.323,-176.320,8.926,148.723
C04949=1161.184,355.603,-79.289,-176.322,8.923,148.722
C04950=1161.189,355.356,-79.254,-176.324,8.919,148.722
C04951=1161.193,355.109,-79.220,-176.327,8.915,148.722
C04952=1161.197,354.861,-79.185,-176.329,8.912,148.721
C04953=1161.200,354.613,-79.152,-176.332,8.908,148.721
C04954=1161.204,354.365,-79.117,-176.334,8.904,148.721
C04955=1161.209,354.118,-79.084,-176.337,8.900,148.721
C04956=1161.213,353.869,-79.049,-176.339,8.897,148.720
C04957=1161.216,353.622,-79.015,-176.342,8.893,148.720
C04958=1161.221,353.375,-78.980,-176.344,8.889,148.720
C04959=1161.224,353.127,-78.946,-176.346,8.886,148.719
C04960=1161.229,352.880,-78.912,-176.349,8.881,148.719
C04961=1161.233,352.633,-78.878,-176.351,8.878,148.719
C04962=1161.237,352.384,-78.844,-176.354,8.875,148.719
C04963=1161.241,352.137,-78.810,-176.356,8.870,148.718
C04964=1161.245,351.889,-78.775,-176.358,8.867,148.718
C04965=1161.249,351.642,-78.741,-176.361,8.863,148.718
C04966=1161.253,351.394,-78.708,-176.364,8.860,148.718
C04967=1161.257,351.146,-78.673,-176.366,8.856,148.717
C04968=1161.260,350.899,-78.639,-176.368,8.852,148.717
C04969=1161.265,350.651,-78.605,-176.371,8.849,148.717
C04970=1161.269,350.403,-78.572,-176.374,8.845,148.716
C04971=1161.272,350.156,-78.537,-176.376,8.841,148.716
C04972=1161.277,349.908,-78.503,-176.378,8.838,148.716
C04973=1161.281,349.660,-78.470,-176.381,8.834,148.716
C04974=1161.285,349.412,-78.435,-176.383,8.830,148.715
C04975=1161.289,349.165,-78.401,-176.386,8.826,148.715
C04976=1161.293,348.918,-78.368,-176.388,8.823,148.715
C04977=1161.297,348.669,-78.333,-176.390,8.820,148.715
C04978=1161.301,348.422,-78.300,-176.393,8.816,148.714
C04979=1161.305,348.175,-78.266,-176.396,8.812,148.714
C04980=1161.309,347.927,-78.233,-176.398,8.809,148.714
C04981=1161.313,347.679,-78.198,-176.401,8.805,148.714
C04982=1161.317,347.431,-78.165,-176.403,8.801,148.713
C04983=1161.321,347.184,-78.131,-176.406,8.797,148.713
C04984=1161.326,346.936,-78.097,-176.408,8.794,148.713
C04985=1161.329,346.688,-78.063,-176.410,8.791,148.713
C04986=1161.333,346.440,-78.030,-176.413,8.786,148.712
C04987=1161.337,346.193,-77.996,-176.415,8.783,148.712
C04988=1161.342,345.945,-77.962,-176.418,8.780,148.712
C04989=1161.346,345.698,-77.928,-176.420,8.776,148.712
C04990=1161.349,345.450,-77.895,-176.423,8.773,148.711
C04991=1161.354,345.202,-77.862,-176.425,8.769,148.711
C04992=1161.358,344.954,-77.827,-176.428,8.765,148.711
C04993=1161.362,344.707,-77.794,-176.430,8.762,148.711
C04994=1161.366,344.460,-77.760,-176.433,8.759,148.711
C04995=1161.370,344.211,-77.727,-176.435,8.754,148.710
C04996=1161.374,343.963,-77.694,-176.437,8.751,148.710
C04997=1161.378,343.716,-77.660,-176.440,8.748,148.710
C04998=1161.382,343.468,-77.626,-176.442,8.743,148.709
C04999=1161.387,343.221,-77.593,-176.445,8.740,148.709
C05000=1161.391,342.973,-77.560,-176.447,8.737,148.709
C05001=1161.394,342.725,-77.525,-176.450,8.733,148.709
C05002=1161.398,342.477,-77.492,-176.452,8.729,148.709
C05003=1161.402,342.230,-77.459,-176.455,8.726,148.708
C05004=1161.406,341.982,-77.426,-176.457,8.722,148.708
C05005=1161.410,341.734,-77.393,-176.460,8.719,148.708
C05006=1161.414,341.487,-77.359,-176.462,8.716,148.708
C05007=1161.419,341.239,-77.325,-176.465,8.711,148.707
C05008=1161.423,340.991,-77.292,-176.467,8.708,148.707
C05009=1161.427,340.743,-77.259,-176.470,8.705,148.707
C05010=1161.431,340.495,-77.225,-176.472,8.701,148.707
C05011=1161.435,340.247,-77.192,-176.475,8.697,148.707
C05012=1161.440,339.968,-77.155,-176.478,8.693,148.706
C05013=1161.444,339.688,-77.117,-176.480,8.689,148.706
C05014=1161.449,339.409,-77.080,-176.483,8.685,148.706
C05015=1161.454,339.129,-77.042,-176.486,8.681,148.706
C05016=1161.458,338.881,-77.009,-176.489,8.678,148.705
C05017=1161.462,338.634,-76.976,-176.491,8.674,148.705
C05018=1161.466,338.386,-76.943,-176.494,8.671,148.705
C05019=1161.470,338.138,-76.909,-176.496,8.667,148.705
C05020=1161.474,337.890,-76.876,-176.499,8.664,148.705
C05021=1161.478,337.642,-76.843,-176.501,8.661,148.704
C05022=1161.482,337.394,-76.810,-176.504,8.657,148.704
C05023=1161.486,337.146,-76.776,-176.506,8.653,148.704
C05024=1161.489,336.899,-76.744,-176.509,8.650,148.704
C05025=1161.494,336.651,-76.711,-176.511,8.647,148.704
C05026=1161.498,336.403,-76.678,-176.514,8.643,148.703
C05027=1161.502,336.155,-76.645,-176.516,8.639,148.703
C05028=1161.506,335.908,-76.612,-176.518,8.636,148.703
C05029=1161.510,335.660,-76.579,-176.521,8.632,148.703
C05030=1161.515,335.412,-76.546,-176.523,8.629,148.702
C05031=1161.519,335.164,-76.513,-176.526,8.625,148.702
C05032=1161.522,334.917,-76.480,-176.529,8.622,148.702
C05033=1161.527,334.669,-76.448,-176.531,8.618,148.702
C05034=1161.531,334.421,-76.414,-176.534,8.615,148.702
C05035=1161.535,334.173,-76.381,-176.536,8.612,148.702
C05036=1161.539,333.925,-76.348,-176.539,8.608,148.701
C05037=1161.543,333.677,-76.316,-176.541,8.604,148.701
C05038=1161.547,333.430,-76.283,-176.543,8.601,148.701
C05039=1161.551,333.182,-76.250,-176.546,8.598,148.701
C05040=1161.556,332.934,-76.218,-176.549,8.594,148.701
C05041=1161.559,332.687,-76.185,-176.551,8.591,148.701
C05042=1161.564,332.439,-76.152,-176.554,8.587,148.700
C05043=1161.568,332.191,-76.120,-176.556,8.584,148.700
C05044=1161.572,331.943,-76.087,-176.559,8.580,148.700
C05045=1161.576,331.696,-76.054,-176.561,8.577,148.700
C05046=1161.580,331.447,-76.022,-176.563,8.573,148.699
C05047=1161.584,331.200,-75.988,-176.566,8.571,148.699
C05048=1161.589,330.951,-75.956,-176.569,8.566,148.699
C05049=1161.592,330.704,-75.923,-176.571,8.563,148.699
C05050=1161.596,330.456,-75.890,-176.574,8.560,148.699
C05051=1161.601,330.208,-75.858,-176.576,8.557,148.699
C05052=1161.605,329.961,-75.826,-176.579,8.552,148.698
C05053=1161.609,329.713,-75.793,-176.582,8.549,148.698
C05054=1161.613,329.465,-75.760,-176.584,8.546,148.698
C05055=1161.617,329.217,-75.728,-176.586,8.543,148.698
C05056=1161.621,328.969,-75.695,-176.589,8.539,148.698
C05057=1161.625,328.721,-75.663,-176.591,8.535,148.698
C05058=1161.629,328.473,-75.630,-176.594,8.533,148.698
C05059=1161.634,328.226,-75.598,-176.596,8.529,148.697
C05060=1161.638,327.978,-75.566,-176.599,8.525,148.697
C05061=1161.642,327.730,-75.533,-176.602,8.522,148.697
C05062=1161.645,327.482,-75.501,-176.604,8.519,148.697
C05063=1161.650,327.234,-75.468,-176.607,8.516,148.697
C05064=1161.654,326.986,-75.435,-176.610,8.511,148.696
C05065=1161.658,326.738,-75.404,-176.612,8.508,148.696
C05066=1161.662,326.491,-75.371,-176.614,8.505,148.696
C05067=1161.666,326.243,-75.339,-176.617,8.502,148.696
C05068=1161.671,325.994,-75.307,-176.619,8.499,148.696
C05069=1161.674,325.746,-75.275,-176.622,8.495,148.696
C05070=1161.679,325.499,-75.242,-176.624,8.491,148.695
C05071=1161.683,325.251,-75.210,-176.627,8.488,148.695
C05072=1161.687,325.003,-75.178,-176.629,8.485,148.695
C05073=1161.691,324.755,-75.145,-176.632,8.481,148.695
C05074=1161.696,324.508,-75.113,-176.635,8.478,148.695
C05075=1161.699,324.260,-75.081,-176.637,8.474,148.695
C05076=1161.704,324.011,-75.049,-176.640,8.471,148.695
C05077=1161.707,323.763,-75.017,-176.642,8.468,148.694
C05078=1161.711,323.515,-74.985,-176.645,8.464,148.694
C05079=1161.716,323.268,-74.952,-176.648,8.461,148.694
C05080=1161.720,323.020,-74.920,-176.650,8.458,148.694
C05081=1161.724,322.772,-74.888,-176.652,8.454,148.694
C05082=1161.728,322.524,-74.856,-176.654,8.451,148.694
C05083=1161.732,322.277,-74.825,-176.658,8.447,148.694
C05084=1161.737,322.028,-74.792,-176.660,8.444,148.693
C05085=1161.740,321.780,-74.760,-176.662,8.441,148.693
C05086=1161.745,321.533,-74.729,-176.665,8.438,148.693
C05087=1161.749,321.284,-74.696,-176.667,8.434,148.693
C05088=1161.753,321.036,-74.665,-176.670,8.430,148.693
C05089=1161.756,320.788,-74.633,-176.673,8.427,148.693
C05090=1161.761,320.541,-74.601,-176.675,8.424,148.693
C05091=1161.765,320.293,-74.569,-176.678,8.421,148.692
C05092=1161.769,320.045,-74.537,-176.680,8.418,148.692
C05093=1161.774,319.797,-74.505,-176.683,8.414,148.692
C05094=1161.778,319.549,-74.473,-176.686,8.410,148.692
C05095=1161.781,319.301,-74.441,-176.688,8.407,148.692
C05096=1161.786,319.053,-74.409,-176.691,8.404,148.692
C05097=1161.790,318.805,-74.377,-176.693,8.401,148.692
C05098=1161.794,318.557,-74.345,-176.695,8.398,148.691
C05099=1161.798,318.310,-74.314,-176.699,8.394,148.691
C05100=1161.803,318.062,-74.281,-176.701,8.391,148.691
C05101=1161.807,317.814,-74.250,-176.703,8.387,148.691
C05102=1161.811,317.566,-74.219,-176.706,8.384,148.691
C05103=1161.815,317.318,-74.187,-176.708,8.381,148.691
C05104=1161.819,317.070,-74.156,-176.710,8.378,148.691
C05105=1161.823,316.822,-74.123,-176.714,8.374,148.691
C05106=1161.828,316.574,-74.092,-176.716,8.371,148.690
C05107=1161.832,316.326,-74.060,-176.719,8.368,148.690
C05108=1161.835,316.078,-74.029,-176.721,8.364,148.690
C05109=1161.840,315.830,-73.997,-176.723,8.361,148.690
C05110=1161.843,315.582,-73.965,-176.726,8.358,148.690
C05111=1161.849,315.334,-73.934,-176.729,8.354,148.690
C05112=1161.852,315.086,-73.902,-176.731,8.351,148.690
C05113=1161.856,314.838,-73.870,-176.734,8.348,148.690
C05114=1161.861,314.590,-73.840,-176.736,8.345,148.689
C05115=1161.864,314.342,-73.808,-176.739,8.342,148.690
C05116=1161.869,314.065,-73.772,-176.742,8.337,148.689
C05117=1161.874,313.788,-73.737,-176.745,8.333,148.689
C05118=1161.879,313.510,-73.702,-176.748,8.330,148.689
C05119=1161.884,313.233,-73.667,-176.751,8.326,148.689
C05120=1161.888,312.985,-73.635,-176.753,8.323,148.689
C05121=1161.892,312.737,-73.604,-176.756,8.320,148.689
C05122=1161.896,312.489,-73.573,-176.758,8.317,148.689
C05123=1161.900,312.241,-73.542,-176.761,8.314,148.688
C05124=1161.904,311.993,-73.510,-176.764,8.310,148.688
C05125=1161.909,311.745,-73.479,-176.766,8.307,148.688
C05126=1161.912,311.497,-73.447,-176.769,8.303,148.688
C05127=1161.917,311.249,-73.417,-176.771,8.300,148.688
C05128=1161.921,311.001,-73.385,-176.774,8.297,148.688
C05129=1161.925,310.753,-73.354,-176.776,8.294,148.688
C05130=1161.929,310.505,-73.322,-176.779,8.291,148.688
C05131=1161.934,310.257,-73.291,-176.781,8.288,148.688
C05132=1161.938,310.009,-73.260,-176.784,8.284,148.688
C05133=1161.942,309.761,-73.229,-176.787,8.281,148.687
C05134=1161.947,309.514,-73.198,-176.789,8.278,148.687
C05135=1161.950,309.265,-73.166,-176.792,8.274,148.687
C05136=1161.955,309.018,-73.135,-176.794,8.271,148.687
C05137=1161.959,308.769,-73.104,-176.797,8.268,148.687
C05138=1161.963,308.522,-73.073,-176.799,8.265,148.687
C05139=1161.967,308.273,-73.042,-176.802,8.262,148.687
C05140=1161.971,308.025,-73.012,-176.805,8.258,148.687
C05141=1161.975,307.778,-72.980,-176.807,8.255,148.687
C05142=1161.979,307.529,-72.949,-176.810,8.251,148.686
C05143=1161.984,307.281,-72.918,-176.812,8.248,148.686
C05144=1161.988,307.033,-72.887,-176.815,8.245,148.686
C05145=1161.992,306.785,-72.856,-176.817,8.242,148.686
C05146=1161.996,306.538,-72.825,-176.820,8.239,148.686
C05147=1162.000,306.289,-72.794,-176.822,8.236,148.686
C05148=1162.005,306.041,-72.763,-176.825,8.233,148.686
C05149=1162.010,305.793,-72.733,-176.828,8.229,148.686
C05150=1162.013,305.545,-72.701,-176.830,8.226,148.686
C05151=1162.018,305.297,-72.670,-176.833,8.223,148.686
C05152=1162.021,305.049,-72.640,-176.835,8.219,148.686
C05153=1162.026,304.801,-72.609,-176.838,8.216,148.686
C05154=1162.030,304.553,-72.578,-176.841,8.213,148.685
C05155=1162.034,304.304,-72.547,-176.843,8.210,148.685
C05156=1162.039,304.056,-72.516,-176.846,8.207,148.685
C05157=1162.043,303.809,-72.486,-176.848,8.204,148.685
C05158=1162.047,303.561,-72.455,-176.851,8.201,148.685
C05159=1162.051,303.312,-72.424,-176.854,8.197,148.685
C05160=1162.055,303.064,-72.394,-176.856,8.193,148.685
C05161=1162.060,302.816,-72.363,-176.859,8.191,148.685
C05162=1162.064,302.568,-72.332,-176.861,8.187,148.685
C05163=1162.069,302.320,-72.301,-176.864,8.184,148.685
C05164=1162.072,302.072,-72.271,-176.867,8.181,148.685
C05165=1162.076,301.823,-72.240,-176.869,8.178,148.685
C05166=1162.081,301.575,-72.209,-176.872,8.175,148.685
C05167=1162.085,301.328,-72.179,-176.874,8.172,148.684
C05168=1162.090,301.080,-72.148,-176.877,8.169,148.685
C05169=1162.094,300.831,-72.117,-176.879,8.165,148.684
C05170=1162.097,300.584,-72.087,-176.882,8.163,148.684
C05171=1162.102,300.336,-72.056,-176.885,8.158,148.684
C05172=1162.107,300.088,-72.025,-176.888,8.155,148.684
C05173=1162.110,299.839,-71.996,-176.890,8.152,148.684
C05174=1162.115,299.591,-71.965,-176.893,8.149,148.684
C05175=1162.119,299.343,-71.935,-176.895,8.146,148.684
C05176=1162.123,299.095,-71.904,-176.898,8.143,148.684
C05177=1162.127,298.847,-71.873,-176.900,8.140,148.684
C05178=1162.131,298.599,-71.843,-176.903,8.137,148.684
C05179=1162.136,298.350,-71.813,-176.905,8.134,148.684
C05180=1162.140,298.103,-71.782,-176.908,8.131,148.684
C05181=1162.145,297.855,-71.752,-176.911,8.127,148.684
C05182=1162.148,297.606,-71.721,-176.913,8.125,148.684
C05183=1162.153,297.358,-71.691,-176.916,8.121,148.683
C05184=1162.157,297.110,-71.661,-176.918,8.118,148.683
C05185=1162.161,296.862,-71.630,-176.921,8.115,148.684
C05186=1162.166,296.614,-71.601,-176.923,8.112,148.683
C05187=1162.170,296.366,-71.570,-176.927,8.108,148.683
C05188=1162.173,296.117,-71.539,-176.929,8.105,148.683
C05189=1162.178,295.869,-71.509,-176.932,8.102,148.683
C05190=1162.182,295.621,-71.479,-176.934,8.099,148.683
C05191=1162.186,295.374,-71.449,-176.937,8.096,148.683
C05192=1162.191,295.125,-71.419,-176.940,8.093,148.683
C05193=1162.195,294.877,-71.389,-176.942,8.089,148.683
C05194=1162.199,294.628,-71.358,-176.945,8.087,148.683
C05195=1162.203,294.380,-71.328,-176.947,8.084,148.683
C05196=1162.208,294.132,-71.298,-176.950,8.080,148.683
C05197=1162.212,293.884,-71.268,-176.952,8.077,148.683
C05198=1162.216,293.636,-71.239,-176.955,8.074,148.683
C05199=1162.221,293.388,-71.208,-176.957,8.071,148.683
C05200=1162.225,293.140,-71.178,-176.960,8.068,148.683
C05201=1162.229,292.892,-71.148,-176.963,8.065,148.683
C05202=1162.234,292.644,-71.118,-176.965,8.062,148.683
C05203=1162.237,292.395,-71.088,-176.968,8.059,148.683
C05204=1162.241,292.147,-71.058,-176.971,8.056,148.683
C05205=1162.246,291.899,-71.027,-176.973,8.053,148.682
C05206=1162.250,291.651,-70.998,-176.976,8.050,148.682
C05207=1162.254,291.402,-70.968,-176.978,8.046,148.682
C05208=1162.259,291.154,-70.938,-176.981,8.043,148.682
C05209=1162.263,290.906,-70.908,-176.984,8.040,148.682
C05210=1162.267,290.659,-70.878,-176.986,8.037,148.682
C05211=1162.272,290.410,-70.848,-176.989,8.034,148.682
C05212=1162.276,290.162,-70.819,-176.991,8.031,148.682
C05213=1162.280,289.913,-70.789,-176.994,8.028,148.682
C05214=1162.284,289.666,-70.759,-176.996,8.025,148.682
C05215=1162.289,289.417,-70.729,-176.999,8.022,148.682
C05216=1162.293,289.169,-70.699,-177.002,8.019,148.682
C05217=1162.297,288.921,-70.669,-177.004,8.016,148.682
C05218=1162.301,288.673,-70.640,-177.007,8.013,148.682
C05219=1162.305,288.425,-70.610,-177.010,8.010,148.682
C05220=1162.310,288.150,-70.577,-177.013,8.006,148.682
C05221=1162.315,287.875,-70.544,-177.015,8.003,148.682
C05222=1162.319,287.600,-70.511,-177.019,7.999,148.682
C05223=1162.324,287.324,-70.478,-177.021,7.996,148.682
C05224=1162.329,287.076,-70.449,-177.024,7.993,148.682
C05225=1162.333,286.828,-70.420,-177.027,7.990,148.682
C05226=1162.337,286.580,-70.389,-177.029,7.987,148.682
C05227=1162.342,286.332,-70.359,-177.032,7.984,148.682
C05228=1162.346,286.083,-70.330,-177.034,7.981,148.682
C05229=1162.350,285.835,-70.300,-177.037,7.978,148.682
C05230=1162.354,285.587,-70.271,-177.040,7.975,148.682
C05231=1162.358,285.339,-70.242,-177.043,7.972,148.682
C05232=1162.362,285.090,-70.212,-177.045,7.968,148.682
C05233=1162.367,284.842,-70.183,-177.048,7.965,148.682
C05234=1162.371,284.595,-70.154,-177.050,7.963,148.682
C05235=1162.376,284.346,-70.124,-177.053,7.960,148.682
C05236=1162.380,284.098,-70.095,-177.055,7.956,148.682
C05237=1162.385,283.849,-70.065,-177.058,7.953,148.682
C05238=1162.389,283.601,-70.035,-177.061,7.950,148.682
C05239=1162.393,283.353,-70.006,-177.064,7.947,148.682
C05240=1162.397,283.105,-69.976,-177.066,7.944,148.682
C05241=1162.401,282.856,-69.947,-177.069,7.941,148.682
C05242=1162.406,282.608,-69.917,-177.072,7.938,148.682
C05243=1162.410,282.361,-69.888,-177.074,7.935,148.682
C05244=1162.415,282.112,-69.859,-177.077,7.932,148.682
C05245=1162.419,281.863,-69.830,-177.079,7.929,148.682
C05246=1162.423,281.615,-69.801,-177.082,7.926,148.682
C05247=1162.427,281.367,-69.771,-177.085,7.923,148.682
C05248=1162.432,281.119,-69.742,-177.087,7.920,148.681
C05249=1162.436,280.870,-69.712,-177.090,7.917,148.682
C05250=1162.440,280.623,-69.684,-177.093,7.914,148.682
C05251=1162.444,280.374,-69.655,-177.095,7.911,148.682
C05252=1162.449,280.126,-69.626,-177.098,7.908,148.682
C05253=1162.453,279.878,-69.596,-177.100,7.905,148.681
C05254=1162.457,279.629,-69.567,-177.103,7.902,148.682
C05255=1162.461,279.380,-69.538,-177.106,7.899,148.682
C05256=1162.466,279.133,-69.509,-177.109,7.896,148.682
C05257=1162.470,278.885,-69.479,-177.111,7.894,148.682
C05258=1162.475,278.636,-69.450,-177.113,7.890,148.682
C05259=1162.478,278.388,-69.422,-177.116,7.887,148.682
C05260=1162.482,278.139,-69.392,-177.119,7.884,148.682
C05261=1162.487,277.892,-69.363,-177.122,7.881,148.682
C05262=1162.492,277.643,-69.334,-177.124,7.879,148.682
C05263=1162.496,277.395,-69.305,-177.127,7.875,148.682
C05264=1162.500,277.146,-69.276,-177.129,7.872,148.682
C05265=1162.504,276.899,-69.248,-177.132,7.869,148.682
C05266=1162.509,276.650,-69.218,-177.135,7.866,148.682
C05267=1162.513,276.401,-69.190,-177.138,7.863,148.682
C05268=1162.517,276.153,-69.160,-177.140,7.860,148.682
C05269=1162.522,275.905,-69.132,-177.143,7.857,148.682
C05270=1162.526,275.657,-69.103,-177.145,7.854,148.682
C05271=1162.530,275.408,-69.074,-177.148,7.851,148.682
C05272=1162.535,275.160,-69.045,-177.151,7.848,148.682
C05273=1162.539,274.912,-69.017,-177.154,7.845,148.682
C05274=1162.543,274.664,-68.988,-177.156,7.842,148.682
C05275=1162.548,274.415,-68.959,-177.159,7.840,148.682
C05276=1162.552,274.167,-68.930,-177.161,7.837,148.682
C05277=1162.556,273.919,-68.902,-177.164,7.834,148.682
C05278=1162.560,273.670,-68.872,-177.166,7.831,148.682
C05279=1162.565,273.422,-68.844,-177.169,7.828,148.682
C05280=1162.569,273.174,-68.815,-177.172,7.825,148.682
C05281=1162.573,272.925,-68.786,-177.175,7.822,148.682
C05282=1162.578,272.677,-68.758,-177.177,7.819,148.682
C05283=1162.582,272.429,-68.729,-177.180,7.816,148.682
C05284=1162.586,272.180,-68.700,-177.183,7.813,148.682
C05285=1162.591,271.932,-68.672,-177.185,7.810,148.682
C05286=1162.595,271.684,-68.643,-177.188,7.807,148.682
C05287=1162.599,271.435,-68.614,-177.190,7.805,148.682
C05288=1162.604,271.188,-68.586,-177.193,7.802,148.682
C05289=1162.608,270.939,-68.557,-177.196,7.799,148.682
C05290=1162.612,270.690,-68.528,-177.198,7.796,148.682
C05291=1162.617,270.442,-68.500,-177.201,7.793,148.682
C05292=1162.621,270.194,-68.472,-177.204,7.790,148.682
C05293=1162.625,269.946,-68.443,-177.206,7.787,148.682
C05294=1162.630,269.697,-68.414,-177.209,7.784,148.682
C05295=1162.634,269.449,-68.386,-177.212,7.781,148.682
C05296=1162.639,269.201,-68.358,-177.215,7.778,148.682
C05297=1162.643,268.952,-68.329,-177.217,7.776,148.682
C05298=1162.647,268.705,-68.301,-177.220,7.773,148.683
C05299=1162.652,268.456,-68.272,-177.222,7.770,148.683
C05300=1162.655,268.207,-68.244,-177.225,7.767,148.683
C05301=1162.660,267.959,-68.215,-177.228,7.764,148.683
C05302=1162.664,267.710,-68.187,-177.231,7.761,148.683
C05303=1162.669,267.462,-68.159,-177.233,7.758,148.683
C05304=1162.673,267.214,-68.131,-177.236,7.755,148.683
C05305=1162.678,266.965,-68.102,-177.239,7.752,148.683
C05306=1162.682,266.717,-68.074,-177.241,7.750,148.683
C05307=1162.686,266.470,-68.046,-177.243,7.747,148.683
C05308=1162.690,266.221,-68.017,-177.246,7.744,148.683
C05309=1162.695,265.973,-67.989,-177.249,7.741,148.683
C05310=1162.699,265.724,-67.961,-177.252,7.738,148.683
C05311=1162.704,265.476,-67.933,-177.254,7.735,148.683
C05312=1162.708,265.227,-67.904,-177.257,7.732,148.683
C05313=1162.712,264.979,-67.876,-177.260,7.729,148.683
C05314=1162.716,264.730,-67.849,-177.262,7.727,148.683
C05315=1162.722,264.482,-67.820,-177.265,7.724,148.683
C05316=1162.725,264.233,-67.792,-177.268,7.721,148.683
C05317=1162.730,263.985,-67.764,-177.270,7.718,148.683
C05318=1162.734,263.737,-67.736,-177.273,7.715,148.683
C05319=1162.738,263.489,-67.708,-177.276,7.712,148.683
C05320=1162.743,263.240,-67.679,-177.279,7.709,148.684
C05321=1162.747,262.992,-67.652,-177.281,7.706,148.684
C05322=1162.751,262.743,-67.623,-177.284,7.704,148.684
C05323=1162.756,262.494,-67.596,-177.286,7.701,148.684
C05324=1162.761,262.222,-67.564,-177.289,7.698,148.684
C05325=1162.765,261.948,-67.534,-177.292,7.694,148.684
C05326=1162.770,261.675,-67.503,-177.295,7.691,148.684
C05327=1162.775,261.402,-67.472,-177.298,7.689,148.684
C05328=1162.779,261.154,-67.445,-177.301,7.686,148.684
C05329=1162.784,260.905,-67.417,-177.303,7.683,148.684
C05330=1162.788,260.657,-67.389,-177.306,7.680,148.684
C05331=1162.793,260.409,-67.361,-177.309,7.677,148.684
C05332=1162.796,260.160,-67.333,-177.311,7.675,148.684
C05333=1162.801,259.912,-67.306,-177.314,7.672,148.684
C05334=1162.806,259.663,-67.277,-177.317,7.669,148.684
C05335=1162.810,259.415,-67.249,-177.319,7.666,148.684
C05336=1162.815,259.166,-67.222,-177.322,7.663,148.685
C05337=1162.818,258.918,-67.194,-177.325,7.660,148.685
C05338=1162.823,258.670,-67.166,-177.328,7.658,148.685
C05339=1162.827,258.421,-67.139,-177.330,7.655,148.685
C05340=1162.832,258.172,-67.110,-177.333,7.652,148.685
C05341=1162.836,257.924,-67.083,-177.336,7.649,148.685
C05342=1162.841,257.676,-67.056,-177.339,7.646,148.685
C05343=1162.845,257.428,-67.027,-177.341,7.643,148.685
C05344=1162.849,257.179,-67.000,-177.344,7.641,148.685
C05345=1162.854,256.931,-66.973,-177.346,7.638,148.685
C05346=1162.858,256.682,-66.945,-177.349,7.635,148.685
C05347=1162.863,256.434,-66.917,-177.352,7.632,148.685
C05348=1162.867,256.185,-66.890,-177.355,7.629,148.686
C05349=1162.871,255.937,-66.862,-177.357,7.627,148.686
C05350=1162.876,255.688,-66.835,-177.360,7.624,148.686
C05351=1162.880,255.440,-66.807,-177.362,7.621,148.686
C05352=1162.884,255.191,-66.779,-177.365,7.618,148.686
C05353=1162.889,254.943,-66.752,-177.368,7.615,148.686
C05354=1162.893,254.695,-66.725,-177.371,7.612,148.686
C05355=1162.898,254.446,-66.697,-177.373,7.611,148.686
C05356=1162.902,254.198,-66.669,-177.376,7.608,148.686
C05357=1162.906,253.949,-66.642,-177.379,7.605,148.686
C05358=1162.911,253.701,-66.614,-177.382,7.602,148.686
C05359=1162.915,253.452,-66.587,-177.384,7.599,148.686
C05360=1162.919,253.204,-66.560,-177.387,7.597,148.687
C05361=1162.924,252.956,-66.532,-177.389,7.594,148.687
C05362=1162.928,252.707,-66.505,-177.392,7.591,148.687
C05363=1162.932,252.458,-66.478,-177.395,7.588,148.687
C05364=1162.937,252.210,-66.450,-177.398,7.585,148.687
C05365=1162.941,251.962,-66.423,-177.400,7.583,148.687
C05366=1162.946,251.713,-66.396,-177.403,7.580,148.687
C05367=1162.951,251.465,-66.369,-177.406,7.577,148.687
C05368=1162.954,251.216,-66.341,-177.409,7.574,148.687
C05369=1162.959,250.968,-66.314,-177.411,7.572,148.687
C05370=1162.964,250.719,-66.286,-177.414,7.569,148.688
C05371=1162.968,250.471,-66.260,-177.416,7.566,148.688
C05372=1162.972,250.222,-66.233,-177.419,7.563,148.688
C05373=1162.976,249.974,-66.205,-177.422,7.560,148.688
C05374=1162.981,249.725,-66.178,-177.424,7.559,148.688
C05375=1162.985,249.477,-66.151,-177.427,7.556,148.688
C05376=1162.990,249.228,-66.124,-177.430,7.553,148.688
C05377=1162.995,248.980,-66.097,-177.433,7.550,148.688
C05378=1162.998,248.731,-66.070,-177.435,7.548,148.688
C05379=1163.003,248.483,-66.043,-177.438,7.545,148.688
C05380=1163.007,248.235,-66.015,-177.440,7.542,148.688
C05381=1163.012,247.986,-65.988,-177.444,7.539,148.689
C05382=1163.016,247.738,-65.961,-177.446,7.537,148.689
C05383=1163.021,247.489,-65.934,-177.449,7.534,148.689
C05384=1163.025,247.241,-65.907,-177.451,7.531,148.689
C05385=1163.029,246.992,-65.880,-177.454,7.528,148.689
C05386=1163.034,246.743,-65.853,-177.456,7.526,148.689
C05387=1163.038,246.495,-65.826,-177.460,7.523,148.689
C05388=1163.042,246.247,-65.799,-177.462,7.520,148.689
C05389=1163.047,245.998,-65.772,-177.465,7.517,148.690
C05390=1163.051,245.750,-65.745,-177.467,7.515,148.690
C05391=1163.056,245.501,-65.718,-177.470,7.512,148.690
C05392=1163.060,245.253,-65.692,-177.473,7.509,148.690
C05393=1163.065,245.004,-65.665,-177.476,7.507,148.690
C05394=1163.070,244.755,-65.638,-177.478,7.505,148.690
C05395=1163.073,244.506,-65.611,-177.481,7.502,148.690
C05396=1163.078,244.258,-65.584,-177.484,7.499,148.690
C05397=1163.082,244.009,-65.557,-177.487,7.496,148.690
C05398=1163.086,243.761,-65.531,-177.489,7.494,148.691
C05399=1163.091,243.513,-65.504,-177.492,7.491,148.691
C05400=1163.096,243.264,-65.477,-177.495,7.488,148.691
C05401=1163.100,243.015,-65.451,-177.498,7.485,148.691
C05402=1163.104,242.767,-65.424,-177.500,7.483,148.691
C05403=1163.109,242.518,-65.397,-177.503,7.480,148.691
C05404=1163.113,242.270,-65.370,-177.506,7.477,148.691
C05405=1163.118,242.022,-65.343,-177.508,7.475,148.691
C05406=1163.122,241.773,-65.317,-177.511,7.472,148.692
C05407=1163.127,241.524,-65.290,-177.513,7.469,148.692
C05408=1163.131,241.276,-65.263,-177.517,7.467,148.692
C05409=1163.135,241.027,-65.238,-177.519,7.465,148.692
C05410=1163.140,240.779,-65.211,-177.522,7.462,148.692
C05411=1163.144,240.531,-65.184,-177.524,7.459,148.692
C05412=1163.149,240.282,-65.157,-177.527,7.457,148.693
C05413=1163.153,240.033,-65.131,-177.530,7.454,148.693
C05414=1163.158,239.785,-65.104,-177.533,7.451,148.693
C05415=1163.163,239.536,-65.078,-177.535,7.448,148.693
C05416=1163.166,239.287,-65.051,-177.538,7.446,148.693
C05417=1163.171,239.039,-65.024,-177.541,7.443,148.693
C05418=1163.175,238.790,-64.999,-177.544,7.440,148.693
C05419=1163.180,238.542,-64.972,-177.546,7.438,148.693
C05420=1163.184,238.293,-64.946,-177.549,7.436,148.694
C05421=1163.189,238.044,-64.919,-177.552,7.433,148.694
C05422=1163.193,237.796,-64.892,-177.554,7.431,148.694
C05423=1163.198,237.548,-64.867,-177.557,7.428,148.694
C05424=1163.202,237.300,-64.840,-177.560,7.425,148.694
C05425=1163.206,237.051,-64.814,-177.562,7.423,148.694
C05426=1163.211,236.802,-64.787,-177.565,7.420,148.694
C05427=1163.215,236.553,-64.761,-177.568,7.417,148.694
C05428=1163.220,236.282,-64.732,-177.571,7.415,148.695
C05429=1163.225,236.010,-64.704,-177.574,7.412,148.695
C05430=1163.230,235.738,-64.674,-177.577,7.409,148.695
C05431=1163.235,235.466,-64.646,-177.580,7.406,148.695
C05432=1163.239,235.218,-64.620,-177.582,7.403,148.695
C05433=1163.244,234.969,-64.594,-177.585,7.401,148.696
C05434=1163.248,234.721,-64.567,-177.588,7.398,148.696
C05435=1163.252,234.472,-64.541,-177.591,7.395,148.696
C05436=1163.258,234.224,-64.515,-177.593,7.393,148.696
C05437=1163.261,233.976,-64.489,-177.596,7.391,148.696
C05438=1163.266,233.726,-64.463,-177.599,7.388,148.696
C05439=1163.271,233.478,-64.437,-177.601,7.386,148.696
C05440=1163.275,233.229,-64.410,-177.604,7.383,148.697
C05441=1163.279,232.981,-64.385,-177.607,7.380,148.697
C05442=1163.284,232.732,-64.358,-177.609,7.378,148.697
C05443=1163.288,232.484,-64.332,-177.612,7.375,148.697
C05444=1163.293,232.235,-64.306,-177.615,7.372,148.697
C05445=1163.297,231.986,-64.280,-177.617,7.370,148.697
C05446=1163.302,231.737,-64.254,-177.621,7.368,148.698
C05447=1163.306,231.488,-64.229,-177.623,7.365,148.698
C05448=1163.310,231.241,-64.203,-177.626,7.363,148.698
C05449=1163.315,230.992,-64.176,-177.629,7.360,148.698
C05450=1163.320,230.743,-64.150,-177.631,7.358,148.698
C05451=1163.324,230.494,-64.125,-177.634,7.355,148.698
C05452=1163.329,230.246,-64.099,-177.637,7.352,148.699
C05453=1163.333,229.998,-64.073,-177.639,7.350,148.699
C05454=1163.338,229.749,-64.046,-177.642,7.347,148.699
C05455=1163.342,229.500,-64.021,-177.645,7.345,148.699
C05456=1163.346,229.251,-63.995,-177.647,7.342,148.699
C05457=1163.351,229.003,-63.970,-177.650,7.340,148.699
C05458=1163.355,228.754,-63.944,-177.653,7.338,148.700
C05459=1163.360,228.505,-63.917,-177.656,7.335,148.700
C05460=1163.364,228.256,-63.892,-177.658,7.332,148.700
C05461=1163.369,228.008,-63.866,-177.661,7.330,148.700
C05462=1163.373,227.760,-63.841,-177.664,7.327,148.700
C05463=1163.378,227.511,-63.815,-177.666,7.325,148.700
C05464=1163.382,227.263,-63.789,-177.669,7.322,148.701
C05465=1163.387,227.014,-63.764,-177.672,7.319,148.701
C05466=1163.391,226.765,-63.738,-177.675,7.318,148.701
C05467=1163.395,226.516,-63.712,-177.677,7.315,148.701
C05468=1163.401,226.268,-63.686,-177.680,7.312,148.701
C05469=1163.405,226.019,-63.660,-177.683,7.310,148.701
C05470=1163.409,225.770,-63.635,-177.686,7.307,148.702
C05471=1163.414,225.522,-63.609,-177.688,7.305,148.702
C05472=1163.418,225.273,-63.584,-177.691,7.302,148.702
C05473=1163.422,225.024,-63.558,-177.693,7.300,148.702
C05474=1163.427,224.776,-63.532,-177.697,7.298,148.702
C05475=1163.431,224.528,-63.507,-177.699,7.295,148.702
C05476=1163.436,224.278,-63.482,-177.702,7.293,148.703
C05477=1163.441,224.030,-63.456,-177.705,7.290,148.703
C05478=1163.445,223.781,-63.431,-177.707,7.288,148.703
